# B&R Automation Studio project PickupStation
Automation Studio 4.12.4.107 SP; technology packages: mapp 5.23.1, mappCockpit 5.23.0, mappMotion 5.23.1, mappView 5.23.0

## Configuration Configuration

CPU X20CP1686X, AutomationRuntime H4.93, Build 4.1.2, Vc V4.73.0

### Task classes (Cpu.sw)
```
Cyclic#1:
  RSModelPic <- RSModelPick.prg
  ConveyorPr <- Source.Conveyor.ConveyorProgram.prg
  StamperPro <- Source.Stamper.StamperProgram.prg
Cyclic#2 (cycle 12000 us, tolerance 12000 us):
  MasterProg <- Source.Master.MasterProgram.prg
  MainMachin <- Source.MainMachine.MainMachineProgram.prg
  PusherProg <- Source.Pusher.PusherProgram.prg
  PickerProg <- Source.Picker.PickerProgram.prg
Cyclic#4:
  Alarms <- Source.Infrastructure.Alarms.Alarms.prg
  HMIProgram <- Source.HMI.HMIProgram.prg
DataObjects: McAcpSys
NcDataObjects: McDriveLog
Binaries: TCLang, McAcpDrv, udbdef, McAcpSim, mvLoader, arflatprv, mCoWebSc, TCData, FWRules, arcoal, arsvcreg, OpcUaSrv, Settings, iomap, asfw, Role, ashwac, sysconf, AxisConfig, arconfig, AlarmsCore, AlarmsHist, TC, ashwd, User, Cam, Users
Libraries: McBase, MpAxis, McAxis, MpBase, McAcpAx, CoTrace, AsZip, FileIO, runtime, MpAlarmX, astime, standard, asstring, MpServer, MpFile, MpUserX, asieccon, asbrstr, dataobj, asepl, asusb, aruser, arssl, sys_lib, powerlnk, arcert, ashw, aseth
```

### Hardware
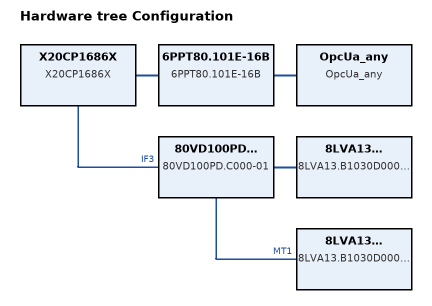
```
6PPT80.101E-16B : 6PPT80.101E-16B v1.0.6.0  [ETH1 -> X20CP1686X.IF2 [Cable Type=PowerlinkCable, Length=10, Version=1.0.0.3]; ETH2 -> OpcUa_any.ETH1 [Cable Type=PowerlinkCable, Length=10, Version=1.0.0.3]]
  Terminal = true
  Startmode = 2
  Mode = Manual
  InternetAddress = 192.168.0.2
  Subnetmask = 255.255.255.0
  ScreenRotation = 180
  PasswordVNC = 
  SelectedFavoriteWeb = 192.168.0.1:81
  BrowserVKeyboard = 0
  PasswordCIFS = 
  PasswordService = 
80VD100PD.C000-01 : 80VD100PD.C000-01 v2.5.0.0  [PLK1 -> X20CP1686X.IF3 (NodeNumber=1) [Cable Type=PowerlinkCable, Length=10, Version=1.0.0.3]; MT2 -> 8LVA13.B1030D000-0.MT]
  DriveConfiguration/Module:
    McAcoposTypeID = AcoposMicroDConfig
    ActivateACOPOSSimulationOnPLC = 1
  DriveConfiguration/Channel[1]/RealAxis:
    AxisReference = gAxisConveyorMpLink
    MechanicalElementsIsInvisible = 0
  DriveConfiguration/Channel[1]/RealAxis/MechanicalElements/Gearbox:
    InputIsReadOnly = 0
    Input = 1
    OutputIsReadOnly = 0
    Output = 1
  DriveConfiguration/Channel[1]/RealAxis/MechanicalElements/RotaryToLinearTransformation:
    ReferenceDistanceIsReadOnly = 0
    ReferenceDistance = 1
  DriveConfiguration/Channel[1]/RealAxis/Controller:
    ModeIsReadOnly = 0
    Mode = PositionController
  DriveConfiguration/Channel[1]/RealAxis/Controller/Mode/Position:
    ProportionalGain = 50.0
    IntegrationTime = 0.0
    PredictionTime = 0.0004
    TotalDelayTime = 0.0004
  DriveConfiguration/Channel[1]/RealAxis/Controller/Mode/Speed:
    ProportionalGainIsReadOnly = 0
    ProportionalGain = 2.0
    IntegrationTimeIsReadOnly = 0
    IntegrationTime = 0.0
    FilterTimeIsReadOnly = 0
    FilterTime = 0.0
  DriveConfiguration/Channel[1]/RealAxis/Controller/Mode/LoopFilters:
    LoopFilterXIsReadOnly = 0
    LoopFilter1 = NotUsed
    LoopFilter2 = NotUsed
    LoopFilter3 = NotUsed
  DriveConfiguration/Channel[1]/RealAxis/Homing:
    ModeIsReadOnly = 0
    Mode = Direct
  DriveConfiguration/Channel[1]/RealAxis/Homing/Mode:
    Position = 0.0
    ReferencePulse = NotUsed
  DriveConfiguration/Channel[1]/RealAxis/Homing:
    RestorePositionVariable = 
  DriveConfiguration/Channel[1]/RealAxis/StopReaction:
    QuickstopIsReadOnly = 0
    Quickstop = DecelerationLimit
    DriveErrorIsReadOnly = 0
    DriveError = DecelerationLimit
  DriveConfiguration/Channel[1]/RealAxis/MovementErrorLimits:
    PositionError = 1.0
    VelocityErrorMonitoring = Automatic1
  DriveConfiguration/Channel[1]/RealAxis:
    JerkFilterIsReadOnly = 0
    JerkFilter = NotUsed
    ZeroVibrationFilter = NotUsed
  DriveConfiguration/Channel[1]/RealAxis/DigitalInputs/HomingSwitch:
    SourceIsReadOnly = 0
    Source = NotUsed
    Level = High
  DriveConfiguration/Channel[1]/RealAxis/DigitalInputs/PositiveLimitSwitch:
    SourceIsReadOnly = 0
    Source = NotUsed
    Level = High
  DriveConfiguration/Channel[1]/RealAxis/DigitalInputs/NegativeLimitSwitch:
    SourceIsReadOnly = 0
    Source = NotUsed
    Level = High
  DriveConfiguration/Channel[1]/RealAxis/DigitalInputs/Trigger1:
    Source = X2Trigger1
    Level = High
  DriveConfiguration/Channel[1]/RealAxis/DigitalInputs/Trigger2:
    Source = X2Trigger2
    Level = High
  DriveConfiguration/Channel[1]/RealAxis/DigitalInputs/Quickstop:
    Input = NotUsed
  DriveConfiguration/Channel[1]/RealAxis/Simulation:
    SimulationModeOnPLC = SetValueGeneration
    SimulationModeOnACOPOS = NotUsed
  DriveConfiguration/Channel[2]/RealAxis:
    AxisReference = gAxisStamperMpLink
    MechanicalElementsIsInvisible = 0
  DriveConfiguration/Channel[2]/RealAxis/MechanicalElements/Gearbox:
    InputIsReadOnly = 0
    Input = 1
    OutputIsReadOnly = 0
    Output = 1
  DriveConfiguration/Channel[2]/RealAxis/MechanicalElements/RotaryToLinearTransformation:
    ReferenceDistanceIsReadOnly = 0
    ReferenceDistance = 1
  DriveConfiguration/Channel[2]/RealAxis/Controller:
    ModeIsReadOnly = 0
    Mode = PositionController
  DriveConfiguration/Channel[2]/RealAxis/Controller/Mode/Position:
    ProportionalGain = 50.0
    IntegrationTime = 0.0
    PredictionTime = 0.0004
    TotalDelayTime = 0.0004
  DriveConfiguration/Channel[2]/RealAxis/Controller/Mode/Speed:
    ProportionalGainIsReadOnly = 0
    ProportionalGain = 2.0
    IntegrationTimeIsReadOnly = 0
    IntegrationTime = 0.0
    FilterTimeIsReadOnly = 0
    FilterTime = 0.0
  DriveConfiguration/Channel[2]/RealAxis/Controller/Mode/LoopFilters:
    LoopFilterXIsReadOnly = 0
    LoopFilter1 = NotUsed
    LoopFilter2 = NotUsed
    LoopFilter3 = NotUsed
  DriveConfiguration/Channel[2]/RealAxis/Homing:
    ModeIsReadOnly = 0
    Mode = Direct
  DriveConfiguration/Channel[2]/RealAxis/Homing/Mode:
    Position = 0.0
    ReferencePulse = NotUsed
  DriveConfiguration/Channel[2]/RealAxis/Homing:
    RestorePositionVariable = 
  DriveConfiguration/Channel[2]/RealAxis/StopReaction:
    QuickstopIsReadOnly = 0
    Quickstop = DecelerationLimit
    DriveErrorIsReadOnly = 0
    DriveError = DecelerationLimit
  DriveConfiguration/Channel[2]/RealAxis/MovementErrorLimits:
    PositionError = 1.0
    VelocityErrorMonitoring = Automatic1
  DriveConfiguration/Channel[2]/RealAxis:
    JerkFilterIsReadOnly = 0
    JerkFilter = NotUsed
    ZeroVibrationFilter = NotUsed
  DriveConfiguration/Channel[2]/RealAxis/DigitalInputs/HomingSwitch:
    SourceIsReadOnly = 0
    Source = NotUsed
    Level = High
  DriveConfiguration/Channel[2]/RealAxis/DigitalInputs/PositiveLimitSwitch:
    SourceIsReadOnly = 0
    Source = NotUsed
    Level = High
  DriveConfiguration/Channel[2]/RealAxis/DigitalInputs/NegativeLimitSwitch:
    SourceIsReadOnly = 0
    Source = NotUsed
    Level = High
  DriveConfiguration/Channel[2]/RealAxis/DigitalInputs/Trigger1:
    Source = X2Trigger1
    Level = High
  DriveConfiguration/Channel[2]/RealAxis/DigitalInputs/Trigger2:
    Source = X2Trigger2
    Level = High
  DriveConfiguration/Channel[2]/RealAxis/DigitalInputs/Quickstop:
    Input = NotUsed
  DriveConfiguration/Channel[2]/RealAxis/Simulation:
    SimulationModeOnPLC = SetValueGeneration
    SimulationModeOnACOPOS = NotUsed
  DriveConfiguration/Channel[2]/RealAxis/AxisFeatures:
    FeatureRef[1] = CamAutomat
8LVA13.B1030D000-0 : 8LVA13.B1030D000-0 v2.2.0.3  [MT -> 80VD100PD.C000-01.MT2]
  M1/MotorParameters:
    MOTOR_AMB_TEMP_RATED = 40
8LVA13.B1030D000-0a : 8LVA13.B1030D000-0 v2.2.0.3  [MT -> 80VD100PD.C000-01.MT1]
  M1/MotorParameters:
    MOTOR_AMB_TEMP_RATED = 40
OpcUa_any : OpcUa_any v1.0.0.1  [ETH1 -> 6PPT80.101E-16B.ETH2 [Cable Type=PowerlinkCable, Length=10, Version=1.0.0.3]]
  ServerEndpointUrl = opc.tcp://192.168.0.3:4840
  Channel1
  ChannelID1 = OUT_HeartBeat
  ChannelBrowsePath1 = /0:Root/0:Objects/4:PLC/4:Modules/6:&:&:/6:Global PV/6:gPickingStation/6:Outputs/6:HeartBeat
  ChannelDirection1 = OUT
  ChannelSamplingInterval1 = 50
  Channel2
  ChannelID2 = OUT_Error
  ChannelBrowsePath2 = /0:Root/0:Objects/4:PLC/4:Modules/6:&:&:/6:Global PV/6:gPickingStation/6:Outputs/6:Error
  ChannelDirection2 = OUT
  ChannelSamplingInterval2 = 50
  Channel3
  ChannelID3 = OUT_WaitingStart
  ChannelBrowsePath3 = /0:Root/0:Objects/4:PLC/4:Modules/6:&:&:/6:Global PV/6:gPickingStation/6:Outputs/6:WaitingStart
  ChannelDirection3 = OUT
  ChannelSamplingInterval3 = 50
  Channel4
  ChannelID4 = OUT_WaitingModeSelection
  ChannelBrowsePath4 = /0:Root/0:Objects/4:PLC/4:Modules/6:&:&:/6:Global PV/6:gPickingStation/6:Outputs/6:WaitingModeSelection
  ChannelDirection4 = OUT
  ChannelSamplingInterval4 = 50
  Channel5
  ChannelID5 = OUT_WaitingInit
  ChannelBrowsePath5 = /0:Root/0:Objects/4:PLC/4:Modules/6:&:&:/6:Global PV/6:gPickingStation/6:Outputs/6:WaitingInit
  ChannelDirection5 = OUT
  ChannelSamplingInterval5 = 50
  Channel6
  ChannelID6 = OUT_InitDone
  ChannelBrowsePath6 = /0:Root/0:Objects/4:PLC/4:Modules/6:&:&:/6:Global PV/6:gPickingStation/6:Outputs/6:InitDone
  ChannelDirection6 = OUT
  ChannelSamplingInterval6 = 50
  Channel7
  ChannelID7 = OUT_Started
  ChannelBrowsePath7 = /0:Root/0:Objects/4:PLC/4:Modules/6:&:&:/6:Global PV/6:gPickingStation/6:Outputs/6:Started
  ChannelDirection7 = OUT
  ChannelSamplingInterval7 = 50
  Channel8
  ChannelID8 = OUT_ClearStatsDone
  ChannelBrowsePath8 = /0:Root/0:Objects/4:PLC/4:Modules/6:&:&:/6:Global PV/6:gPickingStation/6:Outputs/6:ClearStatsDone
  ChannelDirection8 = OUT
  ChannelSamplingInterval8 = 50
  Channel9
  ChannelID9 = OUT_LinkActive
  ChannelBrowsePath9 = /0:Root/0:Objects/4:PLC/4:Modules/6:&:&:/6:Global PV/6:gPickingStation/6:Outputs/6:LinkActive
  ChannelDirection9 = OUT
  ChannelSamplingInterval9 = 50
  Channel10
  ChannelID10 = OUT_ActStampOffset
  ChannelBrowsePath10 = /0:Root/0:Objects/4:PLC/4:Modules/6:&:&:/6:Global PV/6:gPickingStation/6:Outputs/6:ActStampOffset
  ChannelDirection10 = OUT
  ChannelSamplingInterval10 = 50
  ChannelType10 = REAL
  Channel11
  ChannelID11 = OUT_ActStampIncluded
  ChannelBrowsePath11 = /0:Root/0:Objects/4:PLC/4:Modules/6:&:&:/6:Global PV/6:gPickingStation/6:Outputs/6:ActStampIncluded
  ChannelDirection11 = OUT
  ChannelSamplingInterval11 = 50
  Channel12
  ChannelID12 = OUT_CapsOnConveyor
  ChannelBrowsePath12 = /0:Root/0:Objects/4:PLC/4:Modules/6:&:&:/6:Global PV/6:gPickingStation/6:Outputs/6:CapsOnConveyor
  ChannelDirection12 = OUT
  ChannelSamplingInterval12 = 50
  ChannelType12 = USINT
  Channel13
  ChannelID13 = IN_HeartBeat
  ChannelBrowsePath13 = /0:Root/0:Objects/4:PLC/4:Modules/6:&:&:/6:Global PV/6:gPickingStation/6:Inputs/6:HeartBeat
  ChannelPublishingInterval13 = 50
  Channel14
  ChannelID14 = IN_Reset
  ChannelBrowsePath14 = /0:Root/0:Objects/4:PLC/4:Modules/6:&:&:/6:Global PV/6:gPickingStation/6:Inputs/6:Reset
  ChannelPublishingInterval14 = 50
  Channel15
  ChannelID15 = IN_Error
  ChannelBrowsePath15 = /0:Root/0:Objects/4:PLC/4:Modules/6:&:&:/6:Global PV/6:gPickingStation/6:Inputs/6:Error
  ChannelPublishingInterval15 = 50
  Channel16
  ChannelID16 = IN_ClearStats
  ChannelBrowsePath16 = /0:Root/0:Objects/4:PLC/4:Modules/6:&:&:/6:Global PV/6:gPickingStation/6:Inputs/6:ClearStats
  ChannelPublishingInterval16 = 50
  Channel17
  ChannelID17 = IN_Init
  ChannelBrowsePath17 = /0:Root/0:Objects/4:PLC/4:Modules/6:&:&:/6:Global PV/6:gPickingStation/6:Inputs/6:Init
  ChannelPublishingInterval17 = 50
  Channel18
  ChannelID18 = IN_Start
  ChannelBrowsePath18 = /0:Root/0:Objects/4:PLC/4:Modules/6:&:&:/6:Global PV/6:gPickingStation/6:Inputs/6:Start
  ChannelPublishingInterval18 = 50
  Channel19
  ChannelID19 = IN_AutomaticMode
  ChannelBrowsePath19 = /0:Root/0:Objects/4:PLC/4:Modules/6:&:&:/6:Global PV/6:gPickingStation/6:Inputs/6:AutomaticMode
  ChannelPublishingInterval19 = 50
  Channel20
  ChannelID20 = IN_StampIncluded
  ChannelBrowsePath20 = /0:Root/0:Objects/4:PLC/4:Modules/6:&:&:/6:Global PV/6:gPickingStation/6:Inputs/6:StampIncluded
  ChannelPublishingInterval20 = 50
  Channel21
  ChannelID21 = IN_StampOffset
  ChannelBrowsePath21 = /0:Root/0:Objects/4:PLC/4:Modules/6:&:&:/6:Global PV/6:gPickingStation/6:Inputs/6:StampOffset
  ChannelPublishingInterval21 = 50
  ChannelType21 = REAL
  Channel22
  ChannelID22 = IN_ConveyorSpeed
  ChannelBrowsePath22 = /0:Root/0:Objects/4:PLC/4:Modules/6:&:&:/6:Global PV/6:gPickingStation/6:Inputs/6:ConveyorSpeed
  ChannelPublishingInterval22 = 50
  ChannelType22 = REAL
X20CP1686X : X20CP1686X v1.8.0.0
  Connector IF2:
    ActivateDevice = 1
    Mode = Manual
    InternetAddress = 192.168.0.1
    SubnetMask = 255.255.255.0
    ActivateSnmp = 2
  ConfigurationID = PickupStation_Configuration
  VolatileGlobalPvSize = 125535
  TimerDeviceType = EPLX2X
  TimerDevice = X20CP1686X.IF3
  Cyclic1Tolerance = 0
  Cyclic2Duration = 12000
  Cyclic2Tolerance = 12000
  FileDevice1
  FileDeviceName1 = USER
  FileDevicePath1 = USER_PATH
  ActivateOpcUa = 1
  OpcUaInformationModels_PV_Version = 2
  OpcUaInformationModel_Facet = 0
  OpcUaInformationModel_TypeInformation = 0
  OpcUaInformationModel_BaseObjectTypeForStructures = 0
```

### IoMap.iom - X20CP1686X/IoMap.iom
```iecst
VAR_CONFIG
	Cyclic#2.::gMaster.Outputs.HeartBeat AT %IX."OpcUa_any".IN_HeartBeat;
	Cyclic#2.::gMaster.Inputs.HeartBeat AT %QX."OpcUa_any".OUT_HeartBeat;
	Cyclic#2.::gMaster.Inputs.Error AT %QX."OpcUa_any".OUT_Error;
	Cyclic#2.::gMaster.Inputs.WaitingStart AT %QX."OpcUa_any".OUT_WaitingStart;
	Cyclic#2.::gMaster.Inputs.WaitingModeSelection AT %QX."OpcUa_any".OUT_WaitingModeSelection;
	Cyclic#2.::gMaster.Inputs.WaitingInit AT %QX."OpcUa_any".OUT_WaitingInit;
	Cyclic#2.::gMaster.Inputs.InitDone AT %QX."OpcUa_any".OUT_InitDone;
	Cyclic#2.::gMaster.Inputs.Started AT %QX."OpcUa_any".OUT_Started;
	Cyclic#2.::gMaster.Inputs.ClearStatsDone AT %QX."OpcUa_any".OUT_ClearStatsDone;
	Cyclic#2.::gMaster.Outputs.Reset AT %IX."OpcUa_any".IN_Reset;
	Cyclic#2.::gMaster.Outputs.Error AT %IX."OpcUa_any".IN_Error;
	Cyclic#2.::gMaster.Outputs.ClearStats AT %IX."OpcUa_any".IN_ClearStats;
	Cyclic#2.::gMaster.Outputs.Init AT %IX."OpcUa_any".IN_Init;
	Cyclic#2.::gMaster.Outputs.Start AT %IX."OpcUa_any".IN_Start;
	Cyclic#2.::gMaster.Outputs.AutomaticMode AT %IX."OpcUa_any".IN_AutomaticMode;
	Cyclic#2.::gMaster.Outputs.StampIncluded AT %IX."OpcUa_any".IN_StampIncluded;
	Cyclic#2.::gMaster.Outputs.StampOffset AT %ID."OpcUa_any".IN_StampOffset;
	Cyclic#2.::gMaster.Outputs.ConveyorSpeed AT %ID."OpcUa_any".IN_ConveyorSpeed;
	Cyclic#2.::gMainMachine.Commands.OpcuaClientOk AT %IX."OpcUa_any".ModuleOk;
	Cyclic#2.::gMaster.Inputs.LinkActive AT %QX."OpcUa_any".OUT_LinkActive;
	Cyclic#2.::gMaster.Inputs.ActStampOffset AT %QD."OpcUa_any".OUT_ActStampOffset;
	Cyclic#2.::gMaster.Inputs.ActStampIncluded AT %QX."OpcUa_any".OUT_ActStampIncluded;
	::gMaster.Inputs.AskRemoveCaps AT %QX."OpcUa_any".OUT_AskRemoveCaps;
	Cyclic#2.::gMaster.Inputs.CapsOnConveyor AT %QB."OpcUa_any".OUT_CapsOnConveyor;
END_VAR
```

### AxisConfig.axis - X20CP1686X/mappMotion/AxisConfig.axis
```
Element gAxisConveyorMpLink (Type=axis)
  BaseTypeIsReadOnly = 0
  BaseType = LinearPeriodic
    MeasurementUnit = 5066068
    MeasurementResolutionIsReadOnly = 0
    MeasurementResolution = 0.01
    CountDirectionIsReadOnly = 0
    CountDirection = Standard
    PeriodSettings:
      Period = 580
  MovementLimitsIsReadOnly = 0
  MovementLimits = Internal
    Position:
      LowerLimitMin = -1.79769313486231E308
      UpperLimitMax = 1.79769313486231E308
      LowerLimit = -1000.0
      UpperLimit = 1000.0
    VelocityIsReadOnly = 0
    Velocity:
      VelocityMax = 3.4E38
      Velocity = 500
    AccelerationIsReadOnly = 0
    Acceleration:
      AccelerationMax = 3.4E38
      Acceleration = 5000
    DecelerationIsReadOnly = 0
    Deceleration:
      DecelerationMax = 3.4E38
      Deceleration = 5000
  Alarms = MpAlarmX
    mapp.AlarmX.Core.Configuration:
      [2]:
        Severity = 0
Element gAxisStamperMpLink (Type=axis)
  BaseTypeIsReadOnly = 0
  BaseType = Linear
    MeasurementUnit = 5066068
    MeasurementResolutionIsReadOnly = 0
    MeasurementResolution = 0.01
    CountDirectionIsReadOnly = 0
    CountDirection = Standard
  MovementLimitsIsReadOnly = 0
  MovementLimits = Internal
    Position:
      LowerLimitMin = -1.79769313486231E308
      UpperLimitMax = 1.79769313486231E308
      LowerLimit = 0
      UpperLimit = 0.46
    VelocityIsReadOnly = 0
    Velocity:
      VelocityMax = 3.4E38
      Velocity = 100000
    AccelerationIsReadOnly = 0
    Acceleration:
      AccelerationMax = 3.4E38
      Acceleration = 200000
    DecelerationIsReadOnly = 0
    Deceleration:
      DecelerationMax = 3.4E38
      Deceleration = 200000
  Alarms = MpAlarmX
    mapp.AlarmX.Core.Configuration:
      [2]:
        Severity = 0
```

### Cam.axisfeature - X20CP1686X/mappMotion/Cam.axisfeature
```
Element CamAutomat (Type=axisfeature)
  Type = CamAutomat
    CamAutomatType = ACOPOS
      CommonParameters:
        Master:
          ValueSource = SetPosition
            AxisReference = gAxisConveyorMpLink
            MaxVelocity = 500
          StartPosition = 0.0
          StartInterval = MasterAxisPeriod
        AdvancedParameters:
          StartStateParameters:
            StartState = 0
            RelMasterStartPos = 0.0
          AdditiveAxes:
            AdditiveMasterValueSource = NotUsed
            AdditiveSlaveValueSource = NotUsed
          MasterStartPositionMode = NotEvaluatedAnew
          ControlSettings:
            CrossLeftBoundary = PositionLimitedHorizontal
            CamChangeImmediately = CurrentMasterMoveDir
          MessageSettings:
            ErrorsInStandby = NoErrorMessages
          TriggerAndLatch:
            Trigger1Delay = 0.0
            Trigger2Delay = 0.0
            SlaveLatchParID = 0
          EventParIDs
          StartIntervals
          Factors:
            SlaveFactorParID = 0
      States:
        State0 = Used
          Events:
            Event[0]:
              Type = Signal1FromPLC
              Transition = Immediately
              SynchronousUpdate = NotUsed
              NextState = 1
        State[1]:
          Cam = Predefined
            PredefinedCam = OneToOne
          MasterFactor = 20000
          SlaveFactor = 20000
          CompensationMode = DistancesBetweenExitEntryPoints
            MasterDistance = 100
            SlaveDistance = 20
            AdvancedParameters = NotUsed
          AdvancedParameters:
            RepeatCounterInit = 0
            MasterValueSource = CommonMaster
          Events:
            Event[0]:
              Type = StateEnd
              Transition = Immediately
              SynchronousUpdate = NotUsed
              NextState = 2
        State[2]:
          Cam = Predefined
            PredefinedCam = ZeroPoint
          MasterFactor = 1
          SlaveFactor = 0
          CompensationMode = DistancesBetweenExitEntryPoints
            MasterDistance = 100
            SlaveDistance = -220
            AdvancedParameters = NotUsed
          AdvancedParameters:
            RepeatCounterInit = 0
            MasterValueSource = CommonMaster
          Events:
            Event[0]:
              Type = StateEnd
              Transition = Immediately
              SynchronousUpdate = NotUsed
              NextState = 0
```

- Safety project (password-protected, skipped)

### AlarmsCore.mpalarmxcore - X20CP1686X/mappServices/AlarmsCore.mpalarmxcore
```
Element gAlarmXCoreMpLink (Type=mpalarmxcore)
  mapp.AlarmX.Core:
    Mapping:
      [0]
    BySeverity:
      [0]:
        Severity = 1
        [0] = Reaction
          Name = STOP
  mapp.AlarmX.Core.Configuration:
    [0]:
      Name = PickerTimeoutForward
      Message = {$Source/Picker/Alarms/PickerTimeoutForward}
    [1]:
      Name = PickerTimeoutBackward
      Message = {$Source/Picker/Alarms/PickerTimeoutBackward}
    [2]:
      Name = PickerTimeoutVacuumPick
      Message = {$Source/Picker/Alarms/PickerTimeoutVacuumPick}
    [3]:
      Name = PickerTimeoutVacuumPlace
      Message = {$Source/Picker/Alarms/PickerTimeoutVacuumPlace}
    [4]:
      Name = PickerInvalidSensorsCombination
      Message = {$Source/Picker/Alarms/PickerInvalidSensorsCombination}
      Behavior = PersistentAlarm
    [5]:
      Name = PusherTimeoutForward
      Message = {$Source/Pusher/Alarms/PusherTimeoutForward}
    [6]:
      Name = PusherTimeoutBackward
      Message = {$Source/Pusher/Alarms/PusherTimeoutBackward}
    [7]:
      Name = PusherTimeoutMagazineEmpty
      Message = {$Source/Pusher/Alarms/PusherTimeoutMagazineEmpty}
    [8]:
      Name = PusherInvalidSensorsCombination
      Message = {$Source/Pusher/Alarms/PusherInvalidSensorsCombination}
      Behavior = PersistentAlarm
    [9]:
      Name = ConveyorTimeoutHoming
      Message = {$Source/Conveyor/Alarms/ConveyorTimeoutHoming}
    [10]:
      Name = ConveyorTimeoutPowerOn
      Message = {$Source/Conveyor/Alarms/ConveyorTimeoutPowerOn}
    [11]:
      Name = ConveyorMissedCap
      Message = {$Source/Conveyor/Alarms/ConveyorMissedCap}
    [12]:
      Name = ConveyorAxisError
      Message = {$Source/Conveyor/Alarms/ConveyorAxisError}
      Behavior = PersistentAlarm
    [13]:
      Name = ConveyorInitFail
      Message = {$Source/Conveyor/Alarms/ConveyorInitFail}
    [14]:
      Name = ConveyorTooManyCaps
      Message = {$Source/Conveyor/Alarms/ConveyorTooManyCaps}
      Behavior = PersistentAlarm
    [15]:
      Name = StamperAxisError
      Message = {$Source/Stamper/Alarms/StamperAxisError}
      Behavior = PersistentAlarm
    [16]:
      Name = StamperInvalidSensorsCombination
      Message = {$Source/Stamper/Alarms/StamperInvalidSensorsCombination}
      Behavior = PersistentAlarm
    [17]:
      Name = StamperTimeoutHoming
      Message = {$Source/Stamper/Alarms/StamperTimeoutHoming}
    [18]:
      Name = StamperTimeoutPowerOn
      Message = {$Source/Stamper/Alarms/StamperTimeoutPowerOn}
    [19]:
      Name = StamperTimeoutStampBackward
      Message = {$Source/Stamper/Alarms/StamperTimeoutStampBackward}
    [20]:
      Name = StamperTimeoutStampForward
      Message = {$Source/Stamper/Alarms/StamperTimeoutStampForward}
    [21]:
      Name = StamperAxisTimeout
      Message = {$Source/Stamper/Alarms/StamperAxisTimeout}
    [22]:
      Name = MainMachineEmergencyCircuitInterrupted
      Message = {$Source/MainMachine/Alarms/MainMachineEmergencyCircuitInterrupted}
      Behavior = PersistentAlarm
    [23]:
      Name = MainMachineCommunicationLost
      Message = {$Source/MainMachine/Alarms/MainMachineCommunicationLost}
      Behavior = PersistentAlarm
    [24]:
      Name = MainMachineInitializationTimeout
      Message = {$Source/MainMachine/Alarms/MainMachineInitializationTimeout}
    [25]:
      Name = MasterInError
      Message = {$Source/Master/Alarms/MasterInError}
      Behavior:
        MultipleInstances = FALSE
```

### AlarmsHist.mpalarmxhistory - X20CP1686X/mappServices/AlarmsHist.mpalarmxhistory
```
Element gAlarmXHistoryMpLink (Type=mpalarmxhistory)
```

### Users.mpuserx - X20CP1686X/mappServices/Users.mpuserx
```
Element UserMgmtX (Type=mpuserx)
  Mgr:
    LoginAttempts = 0
  ServerSettings:
    Server:
      AdditionalUserData:
        [0] = mail
        [1] = telephoneNumber
  Users:
    DefUser#1:
      id = admin
      name = Andrea Pennisi
      lang = it
      unit = imperial
    DefUser#2:
      id = Anonymous
      lang = en
      unit = metric
  Groups:
    DefGroup#1:
      id = Everyone
      level = 0
    DefGroup#2:
      id = Administrators
      admin = TRUE
```

## Logical view

Binary libraries used (declarations not repeated): operator, runtime, astime, AsIecCon, McBase 5.23.1, MpAxis 5.23.1, McAxis 5.23.1, MpBase 5.23.0, McAcpAx 5.23.1, CoTrace 5.23.0, AsZip, FileIO, MpAlarmX 5.23.1, standard, asstring, MpServer 5.23.0, MpFile 5.23.1, MpUserX 5.23.1


### Program Logical/RSModelPick (IEC) - IO Interface to the RobotStudio model (Pickup IOs)

#### Main.st - Init, cyclic, exit code
```iecst
PROGRAM _INIT
	aiLogoAxisActPos;
	diMagazineEmpty;
	diCapAtPickup;
	diCapPusherForward;
	diCapPusherBack;
	diPickupArmBack;
	diPickupArmForward;
	diCapGripperVacuum;
	diCapOnLogoConveyor;
	diCapExitLogoConveyor;
	diLogoStamperBack;
	diLogoStamperForward;
	aoLogoConveyorSetSpeed;
	doCapPusher;
	doPickupArmForward;
	doPickupArmBack;
	doCapGripperPick;
	aoLogoAxisSetPos;
	doLogoStamper;
	doLogoConveyorClear;

END_PROGRAM

PROGRAM _CYCLIC
	// Pusher
	gPusher.Interface.Inputs.PusherInForwardPosition := diCapPusherForward;
	gPusher.Interface.Inputs.PusherInBackwardPosition := diCapPusherBack;
	gPusher.Interface.Inputs.CapAtPickPosition := diCapAtPickup;
	gPusher.Interface.Inputs.MagazineEmpty := diMagazineEmpty;

	doCapPusher := gPusher.Interface.Outputs.MoveForward;

	// Picker
	gPicker.Interface.Inputs.ArmForward := diPickupArmForward;
	gPicker.Interface.Inputs.ArmBackward := diPickupArmBack;
	gPicker.Interface.Inputs.GripperVacuum := diCapGripperVacuum;

	doPickupArmForward := gPicker.Interface.Outputs.ArmForward;
	doPickupArmBack := gPicker.Interface.Outputs.ArmBackward;
	doCapGripperPick := gPicker.Interface.Outputs.GripperPick;

	// Conveyor
	gConveyor.Interface.Inputs.CapInStartPosition := diCapOnLogoConveyor;
	gConveyor.Interface.Inputs.CapInExitPosition := diCapExitLogoConveyor;

	aoLogoConveyorSetSpeed := gConveyor.Interface.Outputs.SetSpeed/1000;

	// Stamper
	gStamper.Interface.Inputs.ActualPosition := aiLogoAxisActPos*1000;
	gStamper.Interface.Inputs.StampIsForward := diLogoStamperForward;
	gStamper.Interface.Inputs.StampIsBackward := diLogoStamperBack;

	aoLogoAxisSetPos := LREAL_TO_REAL(gStamper.Interface.Outputs.SetPosition/1000);
	doLogoStamper := gStamper.Interface.Outputs.StampForward;
END_PROGRAM

PROGRAM _EXIT

END_PROGRAM
```

#### Variables.var - Local variables
```iecst
(*Inputs*)
VAR
	diMagazineEmpty : BOOL := 0;
	diCapAtPickup : BOOL := 0;
	diCapPusherForward : BOOL := 0;
	diCapPusherBack : BOOL := 0;
	diPickupArmForward : BOOL := 0;
	diPickupArmBack : BOOL := 0;
	diCapGripperVacuum : BOOL := 0;
	diCapOnLogoConveyor : BOOL := 0;
	diLogoStamperForward : BOOL := 0;
	diLogoStamperBack : BOOL := 0;
	diCapExitLogoConveyor : BOOL := 0;
	aiLogoAxisActPos : REAL := 0.0; (*[m]*)
END_VAR
(*Outputs*)
VAR
	doCapPusher : BOOL := 0;
	doPickupArmForward : BOOL := 0;
	doPickupArmBack : BOOL := 0;
	doCapGripperPick : BOOL := 0;
	doLogoStamper : BOOL := 0;
	aoLogoConveyorSetSpeed : REAL := 0.0; (*[m/s]*)
	aoLogoAxisSetPos : REAL := 0.0; (*[m]*)
END_VAR
(*Model Interaction*)
VAR
	doLogoConveyorClear : BOOL := 0;
END_VAR
```

### AlarmsGlobalVariables.var
```iecst
VAR
	gAlarms : AlarmsType;
END_VAR
```

### AlarmsGlobalTypes.typ
```iecst
TYPE
	AlarmsType : 	STRUCT
		Feedbacks : AlarmsFeedbacksType;
		MpAlarmXListUIConnect : MpAlarmXListUIConnectType;
	END_STRUCT;
	AlarmsFeedbacksType : 	STRUCT
		Pendings : UDINT;
	END_STRUCT;
END_TYPE
```

### Program Logical/Source/Infrastructure/Alarms/Alarms (IEC)

#### Main.st - Init, cyclic, exit code
```iecst
PROGRAM _INIT
	// This program is used to manage the machine alarms. Alarms are set/reset in the modules.

	MpAlarmXCoreFB(MpLink := ADR(gAlarmXCoreMpLink), Enable := TRUE);

	MpAlarmXHistoryFB(MpLink := ADR(gAlarmXHistoryMpLink), Enable := TRUE, DeviceName := ADR('ALARMS'));

	MpAlarmXListUIFB(MpLink :=  ADR(gAlarmXCoreMpLink), Enable := TRUE, UIConnect := ADR(gAlarms.MpAlarmXListUIConnect));

END_PROGRAM

PROGRAM _CYCLIC
	MpAlarmXCoreFB();

	MpAlarmXHistoryFB();

	MpAlarmXListUIFB();

	gAlarms.Feedbacks.Pendings := MpAlarmXCoreFB.PendingAlarms;
END_PROGRAM

PROGRAM _EXIT
	MpAlarmXCoreFB.Enable := FALSE;
	MpAlarmXCoreFB();

	MpAlarmXHistoryFB.Enable := FALSE;
	MpAlarmXHistoryFB();

	MpAlarmXListUIFB.Enable := FALSE;
	MpAlarmXListUIFB();

END_PROGRAM
```

#### Variables.var - Local variables
```iecst
VAR
	MpAlarmXCoreFB : MpAlarmXCore;
	MpAlarmXHistoryFB : MpAlarmXHistory;
	MpAlarmXListUIFB : MpAlarmXListUI;
END_VAR
```

### PusherGlobalTypes.typ
```iecst
TYPE
	PusherType : 	STRUCT  (*Pusher Main type*)
		Commands : PusherCommandsType;
		Feedbacks : PusherFeedbacksType;
		Interface : PusherInterfaceType;
	END_STRUCT;
	PusherCommandsType : 	STRUCT
		Enable : BOOL;
		Reset : BOOL;
		Automatic : PusherAutomaticCommandsType;
		Manual : PusherManualCommandsType;
	END_STRUCT;
	PusherFeedbacksType : 	STRUCT  (*Pusher Feedbacks type*)
		Enabled : BOOL;
		Error : BOOL;
		WaitingStart : BOOL;
		CapReady : BOOL;
		WaitingTakeACapCommand : BOOL;
		InitDone : BOOL;
		InitPosition : BOOL;
		TakeACapDone : BOOL;
	END_STRUCT;
	PusherInterfaceType : 	STRUCT  (*Pusher Interface type*)
		Inputs : PusherInterfaceInputsType;
		Outputs : PusherInterfaceOutputsType;
	END_STRUCT;
	PusherInterfaceOutputsType : 	STRUCT  (*Pusher Interface Output type*)
		MoveForward : BOOL;
	END_STRUCT;
	PusherInterfaceInputsType : 	STRUCT  (*Pusher Interface Input type*)
		PusherInBackwardPosition : BOOL;
		PusherInForwardPosition : BOOL;
		CapAtPickPosition : BOOL;
		MagazineEmpty : BOOL;
	END_STRUCT;
	PusherManualCommandsType : 	STRUCT
		Enable : BOOL;
		Push : BOOL;
	END_STRUCT;
	PusherAutomaticCommandsType : 	STRUCT
		Start : BOOL;
		Init : BOOL;
		TakeACap : BOOL;
	END_STRUCT;
END_TYPE
```

### PusherGlobalVariables.var
```iecst
VAR
    gPusher : PusherType;
END_VAR
```

### Program Logical/Source/Pusher/PusherProgram (IEC)

#### Main.st - Init, cyclic, exit code
```iecst
//******************************************************************************************************
// Program: 	PusherProgram
// Author: 		Andrea Pennisi
// Rev.: 		1.0.0
// Date:		5.12.2023
//
// Description:
// This module is used to pick a cap from the magazine station to the pick position.
// Only pneumatic motion in this module
//******************************************************************************************************

PROGRAM _INIT

    ResetOutputsAction;
    ResetFeedbacksAction;

    MachineState.NextState := WAITING_INIT;

END_PROGRAM

PROGRAM _CYCLIC

    // Enable module
    IF NOT gPusher.Commands.Enable THEN
        ResetOutputsAction;
		ResetFeedbacksAction;
		ResetAlarmsAction;
        RETURN;
	END_IF

	IF EDGENEG(gPusher.Commands.Automatic.Start) THEN
		IF MachineState.NextState <> ERROR THEN
			MachineState.NextState := WAITING_START;
		END_IF
	END_IF

	IF EDGEPOS(gPusher.Commands.Automatic.Init) THEN
		IF MachineState.NextState <> ERROR THEN
			MachineState.NextState := WAITING_INIT;
		END_IF
	END_IF

	// Alarms
	SetAlarmsAction;

    // Machine state
    MachineStateManagementAction;
    CASE MachineState.ActualState OF

		WAITING_INIT:
			MachineState.TimeoutTimer.PT := T#0S; // Timeout disabled in this state
			IF MachineState.NewTriggerState THEN
				ResetOutputsAction;
				gPusher.Feedbacks.TakeACapDone := FALSE;
			END_IF
			IF gPusher.Commands.Automatic.Init THEN
				MachineState.NextState := MOVE_BACKWARD;

			ELSIF gPusher.Commands.Manual.Enable THEN
				MachineState.NextState := MANUALS;

			END_IF

		MANUALS:
			MachineState.TimeoutTimer.PT := T#0S; // Timeout disabled in this state
			// Manual commands
			gPusher.Interface.Outputs.MoveForward := gPusher.Commands.Manual.Push;
			IF NOT gPusher.Commands.Manual.Enable THEN
				MachineState.NextState := WAITING_INIT;
			END_IF

		MOVE_BACKWARD:
			MachineState.TimeoutTimer.PT := T#3S;
			IF gPusher.Interface.Inputs.PusherInBackwardPosition THEN
				MachineState.NextState := WAITING_START;
			END_IF

		WAITING_START:
			MachineState.TimeoutTimer.PT := T#0S; // Timeout disabled in this state
			IF gPusher.Commands.Automatic.Start THEN
				MachineState.NextState := WAITING_MAGAZINE;

			ELSIF gPusher.Commands.Manual.Enable THEN
				MachineState.NextState := MANUALS;
			END_IF

		WAITING_MAGAZINE:
			MachineState.TimeoutTimer.PT := T#3S;
			IF NOT gPusher.Interface.Inputs.MagazineEmpty THEN
				MachineState.NextState := WAITING_TAKE_A_CAP_COMMAND;
			END_IF

		WAITING_TAKE_A_CAP_COMMAND:
			MachineState.TimeoutTimer.PT := T#0S; // Timeout disabled in this state
			IF NOT gPusher.Interface.Inputs.CapAtPickPosition AND gPusher.Commands.Automatic.TakeACap THEN
				gPusher.Feedbacks.TakeACapDone := FALSE;
				MachineState.NextState := MOVE_FORWARD;
			END_IF

		MOVE_FORWARD:
			MachineState.TimeoutTimer.PT := T#3S;
			gPusher.Interface.Outputs.MoveForward := TRUE;
			IF gPusher.Interface.Inputs.CapAtPickPosition THEN
				gPusher.Interface.Outputs.MoveForward := FALSE;
				gPusher.Feedbacks.TakeACapDone := TRUE;
				MachineState.NextState := MOVE_BACKWARD;
			END_IF

        ERROR:
			MachineState.TimeoutTimer.PT := T#0S; // Timeout disabled in this state
			ResetOutputsAction;
			IF NOT Internal.Error THEN
				MachineState.NextState := WAITING_INIT;
			END_IF

        ELSE
            MachineState.NextState := WAITING_INIT;

    END_CASE

    FeedbacksUpdateAction;

END_PROGRAM

PROGRAM _EXIT

END_PROGRAM
```

#### Types.typ - Local data types
```iecst
TYPE
	MachineStateType : 	STRUCT  (*Machine state main type*)
		OldState : MachineStateEnum; (*Actual state*)
		ActualState : MachineStateEnum; (*Actual state*)
		NextState : MachineStateEnum; (*Next state*)
		NewTriggerState : BOOL; (*Trigger state change*)
		TimeoutTimer : TON; (*State timeout*)
	END_STRUCT;
	MachineStateEnum :
		( (*Machine State enumeration*)
		WAITING_INIT, (*WAITING state*)
		MANUALS,
		WAITING_START, (*WAITING state*)
		MOVE_BACKWARD,
		WAITING_MAGAZINE, (*ERROR state*)
		WAITING_TAKE_A_CAP_COMMAND,
		MOVE_FORWARD,
		ERROR
		);
	InternalType : 	STRUCT
		Error : BOOL;
	END_STRUCT;
END_TYPE
```

#### Variables.var - Local variables
```iecst
VAR
	MachineState : MachineStateType;
	Internal : InternalType;
END_VAR
```

#### Actions.st
```iecst
ACTION FeedbacksUpdateAction:

	gPusher.Feedbacks.Enabled := TRUE;
    gPusher.Feedbacks.WaitingStart := MachineState.ActualState = WAITING_START;
	gPusher.Feedbacks.Error := MachineState.ActualState = ERROR;
	gPusher.Feedbacks.WaitingTakeACapCommand := MachineState.ActualState = WAITING_TAKE_A_CAP_COMMAND;
	gPusher.Feedbacks.CapReady := gPusher.Interface.Inputs.CapAtPickPosition;
	gPusher.Feedbacks.InitPosition := gPusher.Interface.Inputs.PusherInBackwardPosition;
	gPusher.Feedbacks.InitDone := gPusher.Feedbacks.InitPosition AND gPusher.Commands.Automatic.Init;

END_ACTION

ACTION ResetOutputsAction:

    memset(ADR(gPusher.Interface.Outputs),0,SIZEOF(gPusher.Interface.Outputs));

END_ACTION

ACTION ResetFeedbacksAction:

    memset(ADR(gPusher.Feedbacks),0,SIZEOF(gPusher.Feedbacks));

END_ACTION

ACTION MachineStateManagementAction:

    // Machine state timeout check
    MachineState.TimeoutTimer(IN := MachineState.TimeoutTimer.PT <> T#0S AND NOT MachineState.NewTriggerState);

    // Machine state change state logic
    MachineState.NewTriggerState := (MachineState.ActualState <> MachineState.NextState);
    IF MachineState.NewTriggerState THEN
        MachineState.OldState := MachineState.ActualState;
    END_IF
    MachineState.ActualState := MachineState.NextState;

END_ACTION

ACTION SetAlarmsAction:
	IF gPusher.Commands.Reset THEN
		Internal.Error := FALSE;
	END_IF

    // Timeouts alarms
	IF MachineState.TimeoutTimer.Q THEN
		CASE MachineState.ActualState OF
			MOVE_BACKWARD: MpAlarmXSet(gAlarmXCoreMpLink,'PusherTimeoutBackward'); // Edge alarm!
			MOVE_FORWARD: MpAlarmXSet(gAlarmXCoreMpLink,'PusherTimeoutForward'); // Edge alarm!
			WAITING_MAGAZINE: MpAlarmXSet(gAlarmXCoreMpLink,'PusherTimeoutMagazineEmpty'); // Edge alarm!
		END_CASE
		Internal.Error := TRUE;
		MachineState.NextState := ERROR;
	END_IF

	// PusherInvalidSensorsCombination
	IF gPusher.Interface.Inputs.PusherInBackwardPosition AND gPusher.Interface.Inputs.PusherInForwardPosition THEN
		MpAlarmXSet(gAlarmXCoreMpLink,'PusherInvalidSensorsCombination'); // Periodic alarm!
		Internal.Error := TRUE;
		MachineState.NextState := ERROR;
	ELSE
		MpAlarmXReset(gAlarmXCoreMpLink,'PusherInvalidSensorsCombination');
	END_IF

END_ACTION

ACTION ResetAlarmsAction:

	MpAlarmXReset(gAlarmXCoreMpLink,'PusherInvalidSensorsCombination');

END_ACTION
```

### PickerGlobalTypes.typ
```iecst
TYPE
	PickerType : 	STRUCT  (*Picker Main type*)
		Commands : PickerCommadsType;
		Feedbacks : PickerFeedbacksType;
		Interface : PickerInterfaceType;
	END_STRUCT;
	PickerCommadsType : 	STRUCT  (*Picker Commands type*)
		Enable : BOOL;
		Reset : BOOL;
		Manual : PickerManualCommadsType;
		Automatic : PickerAutomaticCommadsType;
	END_STRUCT;
	PickerFeedbacksType : 	STRUCT  (*Picker Feedbacks type*)
		Enabled : BOOL;
		WaitingPickCommand : BOOL;
		Error : BOOL;
		WaitingStart : BOOL;
		PickACapDone : BOOL;
		InitDone : BOOL;
		InitPosition : BOOL;
	END_STRUCT;
	PickerInterfaceType : 	STRUCT  (*Picker Interface type*)
		Inputs : PickerInterfaceInputsType;
		Outputs : PickerInterfaceOutputsType;
	END_STRUCT;
	PickerInterfaceOutputsType : 	STRUCT  (*Picker Interface Output type*)
		ArmForward : BOOL;
		ArmBackward : BOOL;
		GripperPick : BOOL;
	END_STRUCT;
	PickerInterfaceInputsType : 	STRUCT  (*Picker Interface Input type*)
		ArmBackward : BOOL;
		ArmForward : BOOL;
		GripperVacuum : BOOL;
	END_STRUCT;
	PickerAutomaticCommadsType : 	STRUCT  (*Picker Commands type*)
		PickACap : BOOL;
		Init : BOOL;
		Start : BOOL;
	END_STRUCT;
	PickerManualCommadsType : 	STRUCT  (*Picker Commands type*)
		Enable : BOOL;
		MoveForward : BOOL;
		MoveBackward : BOOL;
		ActivateGrip : BOOL;
	END_STRUCT;
END_TYPE
```

### PickerGlobalVariables.var
```iecst
VAR
    gPicker : PickerType;
END_VAR
```

### Program Logical/Source/Picker/PickerProgram (IEC)

#### Main.st - Init, cyclic, exit code
```iecst
//******************************************************************************************************
// Program: 	PickerProgram
// Author: 		Andrea Pennisi
// Rev.: 		1.0.0
// Date:		5.12.2023
//
// Description:
// This module is used to pick a cap from the pusher station to the conveyor.
// Only pneumatic motion in this module
//******************************************************************************************************

PROGRAM _INIT

    ResetOutputsAction;
    ResetFeedbacksAction;

    MachineState.NextState := WAITING_INIT;

END_PROGRAM

PROGRAM _CYCLIC
    // Enable module
    IF NOT gPicker.Commands.Enable THEN
        ResetOutputsAction;
		ResetFeedbacksAction;
		ResetAlarmsAction;
        RETURN;
    END_IF

	IF EDGENEG(gPicker.Commands.Automatic.Start) THEN
		IF MachineState.NextState <> ERROR THEN
			MachineState.NextState := WAITING_START;
		END_IF
	END_IF

	IF EDGEPOS(gPicker.Commands.Automatic.Init) THEN
		IF MachineState.NextState <> ERROR THEN
			MachineState.NextState := WAITING_INIT;
		END_IF
	END_IF

	// Alarms
	SetAlarmsAction;

    // Machine state
    MachineStateManagementAction;
    CASE MachineState.ActualState OF

		WAITING_INIT:
			MachineState.TimeoutTimer.PT := T#0S; // Timeout disabled in this state
			IF MachineState.NewTriggerState THEN
				ResetOutputsAction;
				gPicker.Feedbacks.PickACapDone := FALSE;
			END_IF

			IF gPicker.Commands.Automatic.Init THEN
				MachineState.NextState := MOVE_BACKWARD;

			ELSIF gPicker.Commands.Manual.Enable THEN
				MachineState.NextState := MANUALS;

			END_IF

		MANUALS:
			MachineState.TimeoutTimer.PT := T#0S; // Timeout disabled in this state
			// Manual commands
			gPicker.Interface.Outputs.ArmForward := gPicker.Commands.Manual.MoveForward;
			gPicker.Interface.Outputs.ArmBackward := gPicker.Commands.Manual.MoveBackward;
			gPicker.Interface.Outputs.GripperPick := gPicker.Commands.Manual.ActivateGrip;

			IF NOT gPicker.Commands.Manual.Enable THEN
				MachineState.NextState := WAITING_INIT;
			END_IF

		MOVE_BACKWARD:
			MachineState.TimeoutTimer.PT := T#3S;
			gPicker.Interface.Outputs.ArmBackward := TRUE;
			IF gPicker.Interface.Inputs.ArmBackward THEN
				gPicker.Interface.Outputs.ArmBackward := FALSE;
				MachineState.NextState := PLACE_CAP;
			END_IF

		PLACE_CAP:
			MachineState.TimeoutTimer.PT := T#3S;
			gPicker.Interface.Outputs.GripperPick := FALSE;
			IF NOT gPicker.Interface.Inputs.GripperVacuum THEN
				gPicker.Feedbacks.PickACapDone := Internal.CapPicked;
				Internal.CapPicked := FALSE;
				MachineState.NextState := WAITING_START;
			END_IF

		WAITING_START:
			MachineState.TimeoutTimer.PT := T#0S; // Timeout disabled in this state
			gPicker.Feedbacks.PickACapDone := FALSE;

			IF gPicker.Commands.Automatic.Start THEN
				MachineState.NextState := WAITING_PICK_COMMAND;

			ELSIF gPicker.Commands.Manual.Enable THEN
				MachineState.NextState := MANUALS;
			END_IF

        WAITING_PICK_COMMAND:
			MachineState.TimeoutTimer.PT := T#0S; // Timeout disabled in this state

			IF gPicker.Commands.Automatic.PickACap THEN
				gPicker.Feedbacks.PickACapDone := FALSE;
                MachineState.NextState := MOVE_FORWARD;
            END_IF

		MOVE_FORWARD:
			MachineState.TimeoutTimer.PT := T#3S;
			gPicker.Interface.Outputs.ArmForward := TRUE;
			IF gPicker.Interface.Inputs.ArmForward THEN
				gPicker.Interface.Outputs.ArmForward := FALSE;
				MachineState.NextState := PICK_CAP;
			END_IF

		PICK_CAP:
			MachineState.TimeoutTimer.PT := T#3S;
			gPicker.Interface.Outputs.GripperPick := TRUE;
			IF gPicker.Interface.Inputs.GripperVacuum THEN
				Internal.CapPicked := TRUE;
				MachineState.NextState := MOVE_BACKWARD;
			END_IF

        ERROR:
            MachineState.TimeoutTimer.PT := T#0S; // Timeout disabled in this state
			ResetOutputsAction;
			IF NOT Internal.Error THEN
				MachineState.NextState := WAITING_INIT;
			END_IF

        ELSE
            MachineState.NextState := WAITING_INIT;

    END_CASE

    FeedbacksUpdateAction;

END_PROGRAM

PROGRAM _EXIT

END_PROGRAM
```

#### Types.typ - Local data types
```iecst
TYPE
	MachineStateType : 	STRUCT  (*Machine state main type*)
		OldState : MachineStateEnum; (*Actual state*)
		ActualState : MachineStateEnum; (*Actual state*)
		NextState : MachineStateEnum; (*Next state*)
		NewTriggerState : BOOL; (*Trigger state change*)
		TimeoutTimer : TON; (*State timeout*)
	END_STRUCT;
	MachineStateEnum :
		( (*Machine State enumeration*)
		WAITING_INIT,
		MANUALS,
		WAITING_START,
		MOVE_BACKWARD, (*INIT state*)
		PLACE_CAP, (*WAITING state*)
		WAITING_PICK_COMMAND, (*ERROR state*)
		MOVE_FORWARD,
		PICK_CAP,
		ERROR
		);
	InternalType : 	STRUCT
		CapPicked : BOOL;
		Error : BOOL;
	END_STRUCT;
END_TYPE
```

#### Variables.var - Local variables
```iecst
VAR
	MachineState : MachineStateType;
	Internal : InternalType;
END_VAR
```

#### Actions.st
```iecst
ACTION FeedbacksUpdateAction:

	gPicker.Feedbacks.Enabled := TRUE;
    gPicker.Feedbacks.WaitingPickCommand := MachineState.ActualState = WAITING_PICK_COMMAND;
    gPicker.Feedbacks.Error := MachineState.ActualState = ERROR;
	gPicker.Feedbacks.InitPosition := gPicker.Interface.Inputs.ArmBackward AND NOT gPicker.Interface.Inputs.GripperVacuum;
	gPicker.Feedbacks.InitDone := gPicker.Feedbacks.InitPosition AND gPicker.Commands.Automatic.Init;

END_ACTION

ACTION ResetOutputsAction:

    memset(ADR(gPicker.Interface.Outputs),0,SIZEOF(gPicker.Interface.Outputs));

END_ACTION

ACTION ResetFeedbacksAction:

    memset(ADR(gPicker.Feedbacks),0,SIZEOF(gPicker.Feedbacks));

END_ACTION

ACTION MachineStateManagementAction:

    // Machine state timeout check
    MachineState.TimeoutTimer(IN := MachineState.TimeoutTimer.PT <> T#0S AND NOT MachineState.NewTriggerState);

	// Machine state change state logic
	MachineState.NewTriggerState := (MachineState.ActualState <> MachineState.NextState);
	IF MachineState.NewTriggerState THEN
		MachineState.OldState := MachineState.ActualState;
	END_IF
	MachineState.ActualState := MachineState.NextState;

END_ACTION

ACTION SetAlarmsAction:

	IF gPicker.Commands.Reset THEN
		Internal.Error := FALSE;
	END_IF

	// Timeouts alarms
	IF MachineState.TimeoutTimer.Q THEN
		CASE MachineState.ActualState OF
			MOVE_BACKWARD: MpAlarmXSet(gAlarmXCoreMpLink,'PickerTimeoutBackward'); // Edge alarm!
			MOVE_FORWARD: MpAlarmXSet(gAlarmXCoreMpLink,'PickerTimeoutForward'); // Edge alarm!
			PLACE_CAP: MpAlarmXSet(gAlarmXCoreMpLink,'PickerTimeoutVacuumPlace'); // Edge alarm!
			PICK_CAP: MpAlarmXSet(gAlarmXCoreMpLink,'PickerTimeoutVacuumPick'); // Edge alarm!
		END_CASE
		Internal.Error := TRUE;
		MachineState.NextState := ERROR;
	END_IF

	// PickupArmInvalidSensorsCombination
	IF gPicker.Interface.Inputs.ArmBackward AND gPicker.Interface.Inputs.ArmForward THEN
		MpAlarmXSet(gAlarmXCoreMpLink,'PickerInvalidSensorsCombination'); // Periodic alarm!
		Internal.Error := TRUE;
		MachineState.NextState := ERROR;
	ELSE
		MpAlarmXReset(gAlarmXCoreMpLink,'PickerInvalidSensorsCombination');
	END_IF

END_ACTION

ACTION ResetAlarmsAction:

	MpAlarmXReset(gAlarmXCoreMpLink,'PickerInvalidSensorsCombination');

END_ACTION
```

### ConveyorGlobalTypes.typ
```iecst
TYPE
	ConveyorType : 	STRUCT  (*Conveyor Main type*)
		Commands : ConveyorCommadsType;
		Feedbacks : ConveyorFeedbacksType;
		Parameters : ConveyorParametersType;
		Interface : ConveyorInterfaceType;
	END_STRUCT;
	ConveyorCommadsType : 	STRUCT  (*Conveyor Commands type*)
		Enable : BOOL;
		Reset : BOOL;
		Automatic : ConveyorAutomaticCommadsType;
		Manual : ConveyorManualCommadsType;
	END_STRUCT;
	ConveyorFeedbacksType : 	STRUCT  (*Conveyor Feedbacks type*)
		Enabled : BOOL;
		WaitingStart : BOOL;
		Error : BOOL;
		WaitingCap : BOOL;
		DeliverCapDone : BOOL;
		InitDone : BOOL;
		AxisHomed : BOOL;
		AxisPowered : BOOL;
		InitPosition : BOOL;
		AxisSpeed : REAL;
		AxisPosition : LREAL;
		CapsOnConveyor : USINT;
	END_STRUCT;
	ConveyorParametersType : 	STRUCT  (*Conveyor Parameters type*)
		TargetSpeed : REAL := 50;
		Acceleration : REAL := 5000;
	END_STRUCT;
	ConveyorInterfaceType : 	STRUCT  (*Conveyor Interface type*)
		Inputs : ConveyorInterfaceInputsType;
		Outputs : ConveyorInterfaceOutputsType;
	END_STRUCT;
	ConveyorInterfaceOutputsType : 	STRUCT  (*Conveyor Interface Output type*)
		SetSpeed : REAL;
	END_STRUCT;
	ConveyorInterfaceInputsType : 	STRUCT  (*Conveyor Interface Input type*)
		CapInStartPosition : BOOL;
		CapInExitPosition : BOOL;
	END_STRUCT;
	ConveyorAutomaticCommadsType : 	STRUCT  (*Conveyor Commands type*)
		Start : BOOL;
		Init : BOOL;
		DeliverCap : BOOL;
	END_STRUCT;
	ConveyorManualCommadsType : 	STRUCT  (*Conveyor Commands type*)
		Enable : BOOL;
		PowerOn : BOOL;
		Move : BOOL;
		Home : BOOL;
		Speed : REAL := 50;
	END_STRUCT;
END_TYPE
```

### ConveyorGlobalVariables.var
```iecst
VAR
    gConveyor : ConveyorType;
END_VAR
```

### Program Logical/Source/Conveyor/ConveyorProgram (IEC)

#### Main.st - Init, cyclic, exit code
```iecst
//******************************************************************************************************
// Program: 	ConveyorProgram
// Author: 		Andrea Pennisi
// Rev.: 		1.0.0
// Date:		5.12.2023
//
// Description:
// This module is used to deliver the cap from the starting position of the conveyor to the exit.
// An axis is controlled by mappMotion tools. The control is made in velocity.
//******************************************************************************************************

PROGRAM _INIT

    ResetOutputsAction;
    ResetFeedbacksAction;

	Internal.Parameters.Homing.Mode := mcHOMING_ABSOLUTE;

    MachineState.NextState := WAITING_INIT;

END_PROGRAM

PROGRAM _CYCLIC

	MotionAction;

    // Enable module
    IF NOT gConveyor.Commands.Enable THEN
        ResetOutputsAction;
		ResetFeedbacksAction;
		ResetAlarmsAction;
		ResetMotionCommands;
        RETURN;
    END_IF

	IF EDGENEG(gConveyor.Commands.Automatic.Start) THEN
		IF MachineState.NextState <> ERROR THEN
			MachineState.NextState := WAITING_START;
		END_IF
	END_IF

	IF EDGEPOS(gConveyor.Commands.Automatic.Init) THEN
		IF MachineState.NextState <> ERROR THEN
			MachineState.NextState := WAITING_INIT;
		END_IF
	END_IF

	// Alarms
	SetAlarmsAction;

    // Machine state
    MachineStateManagementAction;
    CASE MachineState.ActualState OF

		WAITING_INIT:
			MachineState.TimeoutTimer.PT := T#0S; // Timeout disabled in this state
			IF MachineState.NewTriggerState THEN
				ResetOutputsAction;
				ResetMotionCommands;
			END_IF

			IF gConveyor.Commands.Automatic.Init THEN
				gConveyor.Feedbacks.CapsOnConveyor := 0;
				MachineState.NextState := HOMING;

			ELSIF gConveyor.Commands.Manual.Enable THEN
				MachineState.NextState := MANUALS;

			END_IF

		MANUALS:
			MachineState.TimeoutTimer.PT := T#0S; // Timeout disabled in this state

			Internal.Parameters.Velocity := gConveyor.Commands.Manual.Speed;
			IF Internal.Parameters.Velocity>0 THEN
				Internal.Parameters.Direction := mcDIR_POSITIVE;
			ELSE
				Internal.Parameters.Direction := mcDIR_NEGATIVE;
			END_IF

			Internal.Axis.Home := gConveyor.Commands.Manual.Home AND Internal.Axis.Active AND NOT Internal.Axis.Error;
			IF Internal.Axis.IsHomed THEN
				Internal.Axis.Power := gConveyor.Commands.Manual.PowerOn AND Internal.Axis.Active AND NOT Internal.Axis.Error;
				IF Internal.Axis.PowerOn THEN
					Internal.Axis.MoveVelocity := gConveyor.Commands.Manual.Move AND Internal.Axis.Active AND NOT Internal.Axis.Error;
				ELSE
					Internal.Axis.MoveVelocity := FALSE;
				END_IF
			ELSE
				Internal.Axis.Power := FALSE;
				Internal.Axis.MoveVelocity := FALSE;
			END_IF

			IF NOT gConveyor.Commands.Manual.Enable THEN
				MachineState.NextState := WAITING_INIT;
			END_IF

		HOMING:
			MachineState.TimeoutTimer.PT := T#3S;
			IF Internal.Axis.IsHomed THEN
				Internal.Axis.Home := FALSE;
				MachineState.NextState := POWER_ON;
			ELSE
				Internal.Axis.Home := Internal.Axis.Active AND NOT Internal.Axis.Error;
			END_IF

		POWER_ON:
			MachineState.TimeoutTimer.PT := T#3S;
			Internal.Axis.Power := Internal.Axis.Active AND NOT Internal.Axis.Error;
			IF Internal.Axis.PowerOn THEN
				IF gConveyor.Commands.Automatic.Init THEN
					MachineState.NextState := INIT;
				ELSE
					MachineState.NextState := WAITING_CAP;
				END_IF
			END_IF

		INIT:
			MachineState.TimeoutTimer.PT := T#30S;
			IF MachineState.NewTriggerState THEN
				Internal.Parameters.Velocity := gConveyor.Parameters.TargetSpeed;
				Internal.Parameters.Direction := mcDIR_POSITIVE;
			END_IF
			Internal.Axis.MoveAbsolute := Internal.Axis.Active AND NOT Internal.Axis.Error;
			IF Internal.Axis.MoveDone THEN
				Internal.Axis.MoveAbsolute := FALSE;
				MachineState.NextState := WAITING_START;
			END_IF

        WAITING_START:
			MachineState.TimeoutTimer.PT := T#0S; // Timeout disabled in this state
			IF MachineState.NewTriggerState THEN
				Internal.Axis.Power := FALSE;
			END_IF
			gConveyor.Feedbacks.DeliverCapDone := FALSE;
            IF gConveyor.Commands.Automatic.Start THEN
				MachineState.NextState := POWER_ON;

			ELSIF gConveyor.Commands.Manual.Enable THEN
				MachineState.NextState := MANUALS;
            END_IF

		WAITING_CAP:
			MachineState.TimeoutTimer.PT := T#0S; // Timeout disabled in this state
			IF gConveyor.Interface.Inputs.CapInStartPosition AND gConveyor.Commands.Automatic.DeliverCap THEN
				gConveyor.Feedbacks.DeliverCapDone := FALSE;
				MachineState.NextState := MOTION;
			END_IF

		MOTION:
			MachineState.TimeoutTimer.PT := T#30S;
			IF MachineState.NewTriggerState THEN
				Internal.Parameters.Direction := mcDIR_POSITIVE;
			END_IF

			// On-fly velocity change
			IF Internal.Parameters.Velocity <> gConveyor.Parameters.TargetSpeed THEN
				Internal.Parameters.Velocity := gConveyor.Parameters.TargetSpeed;
				Internal.Axis.Update := TRUE;
			ELSIF Internal.Axis.UpdateDone THEN
				Internal.Axis.Update := FALSE;
			END_IF

			Internal.Axis.MoveVelocity := TRUE;
			IF EDGENEG(gConveyor.Interface.Inputs.CapInExitPosition) THEN
				gConveyor.Feedbacks.DeliverCapDone := TRUE;
				Internal.Axis.MoveVelocity := FALSE;
				Internal.Axis.Update := FALSE;
				MachineState.NextState := WAITING_CAP;
			END_IF

        ERROR:
            MachineState.TimeoutTimer.PT := T#0S; // Timeout disabled in this state
			ResetOutputsAction;
			ResetMotionCommands;
			IF NOT Internal.Error THEN
				MachineState.NextState := WAITING_INIT;
			END_IF

        ELSE
            MachineState.NextState := WAITING_START;

    END_CASE

    FeedbacksUpdateAction;

END_PROGRAM

PROGRAM _EXIT

END_PROGRAM
```

#### Types.typ - Local data types
```iecst
TYPE
	MachineStateType : 	STRUCT  (*Machine state main type*)
		OldState : MachineStateEnum; (*Actual state*)
		ActualState : MachineStateEnum; (*Actual state*)
		NextState : MachineStateEnum; (*Next state*)
		NewTriggerState : BOOL; (*Trigger state change*)
		TimeoutTimer : TON; (*State timeout*)
	END_STRUCT;
	MachineStateEnum :
		( (*Machine State enumeration*)
		WAITING_INIT, (*WAITING state*)
		MANUALS,
		WAITING_START,
		HOMING,
		POWER_ON,
		INIT,
		WAITING_CAP,
		MOTION,
		ERROR (*ERROR state*)
		);
	InternalType : 	STRUCT
		Axis : MpAxisBasic;
		Parameters : MpAxisBasicParType;
		Error : BOOL;
	END_STRUCT;
END_TYPE
```

#### Variables.var - Local variables
```iecst
VAR
	MachineState : MachineStateType;
	Internal : InternalType;
END_VAR
```

#### Actions.st
```iecst
ACTION FeedbacksUpdateAction:

    gConveyor.Feedbacks.Enabled := TRUE;
    gConveyor.Feedbacks.WaitingStart := MachineState.ActualState = WAITING_START;
    gConveyor.Feedbacks.Error := MachineState.ActualState = ERROR;
	gConveyor.Feedbacks.WaitingCap := MachineState.ActualState = WAITING_CAP;
	gConveyor.Feedbacks.AxisHomed := Internal.Axis.IsHomed;
	gConveyor.Feedbacks.AxisPowered := Internal.Axis.PowerOn;
	gConveyor.Feedbacks.InitPosition := ABS(Internal.Axis.Position - Internal.Parameters.Position)<0.1;
	gConveyor.Feedbacks.InitDone := gConveyor.Feedbacks.InitPosition AND gConveyor.Commands.Automatic.Init;
	gConveyor.Feedbacks.AxisSpeed := Internal.Axis.Velocity;
	gConveyor.Feedbacks.AxisPosition := Internal.Axis.Position;

	IF EDGEPOS(gConveyor.Interface.Inputs.CapInStartPosition) AND gConveyor.Commands.Automatic.Start THEN
		gConveyor.Feedbacks.CapsOnConveyor := gConveyor.Feedbacks.CapsOnConveyor + 1;

	ELSIF gConveyor.Interface.Inputs.CapInStartPosition AND gConveyor.Commands.Automatic.Start AND gConveyor.Feedbacks.CapsOnConveyor = 0 THEN
		gConveyor.Feedbacks.CapsOnConveyor := gConveyor.Feedbacks.CapsOnConveyor + 1;
	END_IF

	IF EDGEPOS(gConveyor.Interface.Inputs.CapInExitPosition) THEN
		IF gConveyor.Feedbacks.CapsOnConveyor>1 THEN
			gConveyor.Feedbacks.CapsOnConveyor := gConveyor.Feedbacks.CapsOnConveyor - 1;
		ELSE
			gConveyor.Feedbacks.CapsOnConveyor := 0;
		END_IF
	END_IF

END_ACTION

ACTION ResetOutputsAction:

	memset(ADR(gConveyor.Interface.Outputs),0,SIZEOF(gConveyor.Interface.Outputs));

END_ACTION

ACTION ResetMotionCommands:
	Internal.Axis.Power := FALSE;
	Internal.Axis.Home := FALSE;
	Internal.Axis.MoveVelocity := FALSE;
	Internal.Axis.MoveAbsolute := FALSE;
	Internal.Axis.Update := FALSE;
END_ACTION

ACTION ResetFeedbacksAction:

    memset(ADR(gConveyor.Feedbacks),0,SIZEOF(gConveyor.Feedbacks));

END_ACTION

ACTION MachineStateManagementAction:

    // Machine state timeout check
    MachineState.TimeoutTimer(IN := MachineState.TimeoutTimer.PT <> T#0S AND NOT MachineState.NewTriggerState);

    // Machine state change state logic
    MachineState.NewTriggerState := (MachineState.ActualState <> MachineState.NextState);
    IF MachineState.NewTriggerState THEN
        MachineState.OldState := MachineState.ActualState;
    END_IF
    MachineState.ActualState := MachineState.NextState;

END_ACTION

ACTION SetAlarmsAction:

	IF gConveyor.Commands.Reset THEN
		Internal.Error := FALSE;
	END_IF

	// Timeouts
	IF MachineState.TimeoutTimer.Q THEN

		CASE MachineState.ActualState OF
			HOMING: MpAlarmXSet(gAlarmXCoreMpLink,'ConveyorTimeoutHoming'); // Edge alarm!
			POWER_ON: MpAlarmXSet(gAlarmXCoreMpLink,'ConveyorTimeoutPowerOn'); // Edge alarm!
			MOTION: MpAlarmXSet(gAlarmXCoreMpLink,'ConveyorMissedCap'); // Edge alarm!
			INIT: MpAlarmXSet(gAlarmXCoreMpLink,'ConveyorInitFail'); // Edge alarm!
		END_CASE

		Internal.Error := TRUE;
		MachineState.NextState := ERROR;
	END_IF

	// ConveyorAxisError
	IF Internal.Axis.Error THEN
		MpAlarmXSet(gAlarmXCoreMpLink,'ConveyorAxisError');
		Internal.Error := TRUE;
		MachineState.NextState := ERROR;
	ELSE
		MpAlarmXReset(gAlarmXCoreMpLink,'ConveyorAxisError');
	END_IF

	// ConveyorTooManyCaps
	IF gConveyor.Commands.Reset THEN
		gConveyor.Feedbacks.CapsOnConveyor := 0;
	END_IF
	IF gConveyor.Feedbacks.CapsOnConveyor > 1 THEN
		MpAlarmXSet(gAlarmXCoreMpLink,'ConveyorTooManyCaps');
		Internal.Error := TRUE;
		MachineState.NextState := ERROR;
	ELSE
		MpAlarmXReset(gAlarmXCoreMpLink,'ConveyorTooManyCaps');
	END_IF
END_ACTION

ACTION ResetAlarmsAction:

	MpAlarmXReset(gAlarmXCoreMpLink,'ConveyorAxisError');

END_ACTION
```

#### MotionAction.ld
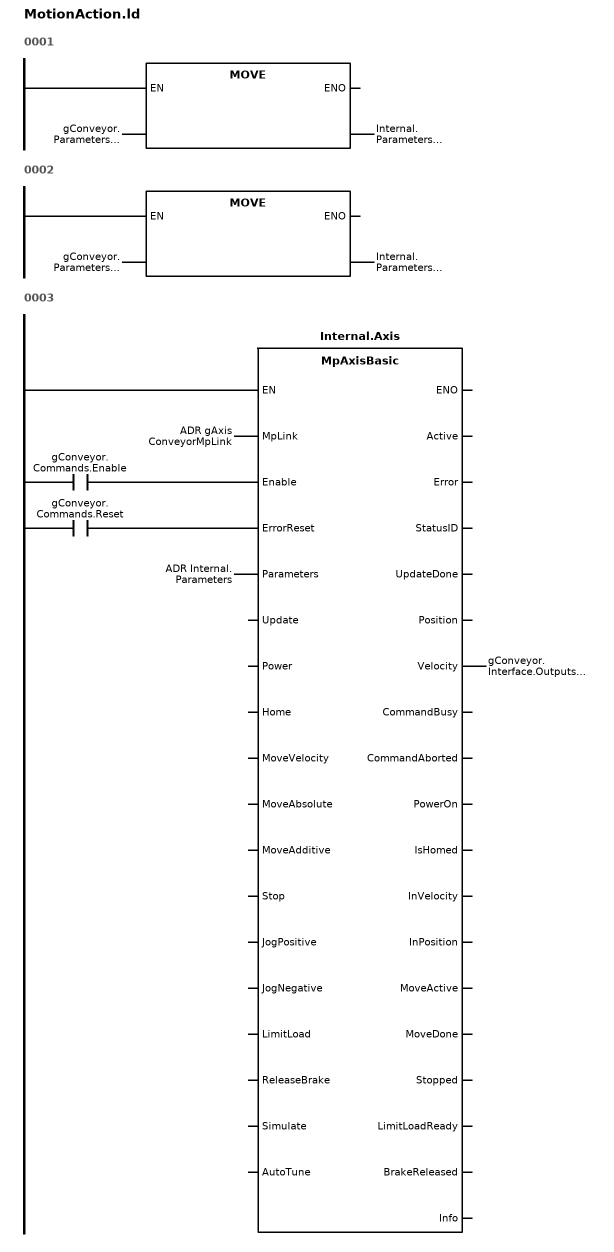
Ladder, written as Structured Text:
```iecst
ACTION MotionAction:
(* Network 1 *)
Internal.Parameters.Deceleration := gConveyor.Parameters.Acceleration;

(* Network 2 *)
Internal.Parameters.Acceleration := gConveyor.Parameters.Acceleration;

(* Network 3 *)
Internal.Axis(MpLink := ADR(gAxisConveyorMpLink), Enable := gConveyor.Commands.Enable, ErrorReset := gConveyor.Commands.Reset, Parameters := ADR(Internal.Parameters));
gConveyor.Interface.Outputs.SetSpeed := Internal.Axis.Velocity;
END_ACTION
```

### StamperGlobalTypes.typ
```iecst
TYPE
	StamperType : 	STRUCT  (*Stamper Main type*)
		Commands : StamperCommadsType;
		Feedbacks : StamperFeedbacksType;
		Parameters : StamperParametersType;
		Interface : StamperInterfaceType;
	END_STRUCT;
	StamperCommadsType : 	STRUCT  (*Stamper Commands type*)
		Enable : BOOL;
		Reset : BOOL;
		Automatic : StamperAutomaticCommadsType;
		Manual : StamperManualCommadsType;
	END_STRUCT;
	StamperFeedbacksType : 	STRUCT  (*Stamper Feedbacks type*)
		Enabled : BOOL;
		WaitingStart : BOOL;
		Error : BOOL;
		OnSyncMotion : BOOL;
		WaitingCap : BOOL;
		StampCapDone : BOOL;
		InitDone : BOOL;
		InitPosition : BOOL;
		AxisSpeed : REAL;
		AxisPosition : LREAL;
		AxisHomed : BOOL;
		AxisPowered : BOOL;
	END_STRUCT;
	StamperParametersType : 	STRUCT  (*Stamper Parameters type*)
		Offset : REAL := 65;
		Speed : REAL := 10000;
		Acceleration : REAL := 20000;
	END_STRUCT;
	StamperInterfaceType : 	STRUCT  (*Stamper Interface type*)
		Inputs : StamperInterfaceInputsType;
		Outputs : StamperInterfaceOutputsType;
	END_STRUCT;
	StamperInterfaceOutputsType : 	STRUCT  (*Stamper Interface Output type*)
		StampForward : BOOL;
		SetPosition : LREAL;
	END_STRUCT;
	StamperInterfaceInputsType : 	STRUCT  (*Stamper Interface Input type*)
		ActualPosition : REAL;
		StampIsForward : BOOL;
		StampIsBackward : BOOL;
	END_STRUCT;
	StamperAutomaticCommadsType : 	STRUCT  (*Stamper Commands type*)
		Start : BOOL;
		Init : BOOL;
		StampCap : BOOL;
	END_STRUCT;
	StamperManualCommadsType : 	STRUCT  (*Stamper Commands type*)
		Enable : BOOL;
		StamperForward : BOOL;
		Position : LREAL;
		Speed : REAL := 50;
		PowerOn : BOOL;
		Move : BOOL;
		Home : BOOL;
	END_STRUCT;
END_TYPE
```

### StamperGlobalVariables.var
```iecst
VAR
    gStamper : StamperType;
END_VAR
```

### Program Logical/Source/Stamper/StamperProgram (IEC)

#### Main.st - Init, cyclic, exit code
```iecst
//******************************************************************************************************
// Program: 	StamperProgram
// Author: 		Andrea Pennisi
// Rev.: 		1.0.0
// Date:		5.12.2023
//
// Description:
// This module is used to stamp the logo in the cap.
// An axis is controlled by mappMotion tools. The control is made by a cam linked to the Conveyor module axis.
//******************************************************************************************************
PROGRAM _INIT

    ResetOutputsAction;
    ResetFeedbacksAction;

	Internal.Parameters.Homing.Mode := mcHOMING_DIRECT;

	Internal.Offset.AdvancedParameters.ShiftMode := mcSHIFT_ABSOLUTE;
	Internal.Offset.Enable := TRUE;

    MachineState.NextState := WAITING_INIT;

END_PROGRAM

PROGRAM _CYCLIC

	MotionAction;

    // Enable module
    IF NOT gStamper.Commands.Enable THEN
        ResetOutputsAction;
		ResetFeedbacksAction;
		ResetAlarmsAction;
		ResetMotionCommands;
        RETURN;
    END_IF

	IF EDGENEG(gStamper.Commands.Automatic.Start) THEN
		IF MachineState.NextState <> ERROR THEN
			MachineState.NextState := WAITING_START;
		END_IF
	END_IF

	IF EDGEPOS(gStamper.Commands.Automatic.Init) THEN
		IF MachineState.NextState <> ERROR THEN
			MachineState.NextState := WAITING_INIT;
		END_IF
	END_IF

	// Alarms
	SetAlarmsAction;

    // Machine state
    MachineStateManagementAction;
    CASE MachineState.ActualState OF

		WAITING_INIT:
			MachineState.TimeoutTimer.PT := T#0S; // Timeout disabled in this state
			IF MachineState.NewTriggerState THEN
				ResetOutputsAction;
				ResetMotionCommands;
				Internal.CamStartTrigger := FALSE;
			END_IF

			IF gStamper.Commands.Automatic.Init THEN
				MachineState.NextState := HOMING;

			ELSIF gStamper.Commands.Manual.Enable THEN
				MachineState.NextState := MANUAL;

			END_IF

		MANUAL:
			MachineState.TimeoutTimer.PT := T#0S; // Timeout disabled in this state

			Internal.Parameters.Velocity := gStamper.Commands.Manual.Speed;
			Internal.Parameters.Position := gStamper.Commands.Manual.Position;

			gStamper.Interface.Outputs.StampForward := gStamper.Commands.Manual.StamperForward;

			Internal.Axis.Home := gStamper.Commands.Manual.Home AND Internal.Axis.Active AND NOT Internal.Axis.Error;
			IF Internal.Axis.IsHomed THEN
				Internal.Axis.Power := gStamper.Commands.Manual.PowerOn AND Internal.Axis.Active AND NOT Internal.Axis.Error;
				IF Internal.Axis.PowerOn THEN
					Internal.Axis.MoveAbsolute := gStamper.Commands.Manual.Move AND Internal.Axis.Active AND NOT Internal.Axis.Error;
				ELSE
					Internal.Axis.MoveAbsolute := FALSE;
				END_IF
			ELSE
				Internal.Axis.Power := FALSE;
				Internal.Axis.MoveAbsolute := FALSE;
			END_IF

			IF NOT gStamper.Commands.Manual.Enable THEN
				MachineState.NextState := WAITING_INIT;
			END_IF

		HOMING:
			MachineState.TimeoutTimer.PT := T#3S;
			IF Internal.Axis.IsHomed THEN
				Internal.Axis.Home := FALSE;
				MachineState.NextState := POWER_ON;
			ELSE
				Internal.Axis.Home := Internal.Axis.Active AND NOT Internal.Axis.Error;
			END_IF

		POWER_ON:
			MachineState.TimeoutTimer.PT := T#3S;

			Internal.Axis.Power := Internal.Axis.Active AND NOT Internal.Axis.Error;
			IF Internal.Axis.PowerOn THEN
				IF gStamper.Commands.Automatic.Init THEN
					MachineState.NextState := INIT;
				ELSE
					MachineState.NextState := ACTIVATE_CAM;
				END_IF
			END_IF

		INIT:
			MachineState.TimeoutTimer.PT := T#15S;
			Internal.Parameters.Velocity := gStamper.Parameters.Speed;
			Internal.Parameters.Position := 0;
			Internal.Axis.MoveAbsolute := Internal.Axis.Active AND NOT Internal.Axis.Error;
			IF Internal.Axis.MoveDone THEN
				Internal.OffsetToDo := TRUE;
				Internal.Axis.MoveAbsolute := FALSE;
				MachineState.NextState := WAITING_START;
			END_IF

        WAITING_START:
			MachineState.TimeoutTimer.PT := T#0S; // Timeout disabled in this state
			IF MachineState.NewTriggerState THEN
				ResetMotionCommands;
				Internal.Parameters.Velocity := gStamper.Parameters.Speed;
			END_IF

			IF gStamper.Commands.Automatic.Start THEN
				gStamper.Feedbacks.StampCapDone := FALSE;
				MachineState.NextState := POWER_ON;

			ELSIF gStamper.Commands.Manual.Enable THEN
				MachineState.NextState := MANUAL;
            END_IF

		ACTIVATE_CAM:
			MachineState.TimeoutTimer.PT := T#0S; // Timeout disabled in this state
			Internal.Cam.Enable := TRUE;
			Internal.Cam.Start := TRUE;
			IF Internal.Axis.Info.PLCopenState = mcAXIS_SYNCHRONIZED_MOTION THEN
				MachineState.NextState := WAITING_CAP;
			END_IF

		WAITING_CAP:
			MachineState.TimeoutTimer.PT := T#0S; // Timeout disabled in this state
			IF gStamper.Commands.Automatic.StampCap THEN
				gStamper.Feedbacks.StampCapDone := FALSE;
				Internal.CamStartTrigger := TRUE;
			END_IF

			IF Internal.Cam.InCam AND Internal.Cam.ActualStateIndex = 1 THEN // Syncronized motion
				Internal.CamStartTrigger := FALSE;
				MachineState.NextState := STAMP_FORWARD;
			END_IF

		STAMP_FORWARD:
			MachineState.TimeoutTimer.PT := T#3S;

			gStamper.Interface.Outputs.StampForward := TRUE;
			IF gStamper.Interface.Inputs.StampIsForward THEN
				MachineState.NextState := STAMPING;
			END_IF

		STAMPING:
			MachineState.TimeoutTimer.PT := T#15S;

			IF Internal.Cam.ActualStateIndex <> 1 THEN
				gStamper.Interface.Outputs.StampForward := FALSE;
				MachineState.NextState := STAMP_BACKWARD;
			END_IF

		STAMP_BACKWARD:
			MachineState.TimeoutTimer.PT := T#3S;

			IF gStamper.Interface.Inputs.StampIsBackward THEN
				gStamper.Feedbacks.StampCapDone := TRUE;
				MachineState.NextState := WAITING_CAP;
			END_IF

        ERROR:
            MachineState.TimeoutTimer.PT := T#0S; // Timeout disabled in this state
			ResetOutputsAction;
			ResetMotionCommands;
			IF NOT Internal.Error THEN
				MachineState.NextState := WAITING_INIT;
			END_IF

        ELSE
            MachineState.NextState := WAITING_START;

    END_CASE

	OffsetManagement;

    FeedbacksUpdateAction;

END_PROGRAM

PROGRAM _EXIT

END_PROGRAM
```

#### Types.typ - Local data types
```iecst
TYPE
	MachineStateType : 	STRUCT  (*Machine state main type*)
		OldState : MachineStateEnum; (*Actual state*)
		ActualState : MachineStateEnum; (*Actual state*)
		NextState : MachineStateEnum; (*Next state*)
		NewTriggerState : BOOL; (*Trigger state change*)
		TimeoutTimer : TON; (*State timeout*)
	END_STRUCT;
	MachineStateEnum :
		( (*Machine State enumeration*)
		WAITING_INIT,
		MANUAL,
		WAITING_START, (*WAITING state*)
		HOMING,
		POWER_ON, (*INIT state*)
		INIT,
		ACTIVATE_CAM,
		WAITING_CAP,
		STAMP_FORWARD,
		STAMPING,
		STAMP_BACKWARD,
		ERROR (*ERROR state*)
		);
	InternalType : 	STRUCT
		Axis : MpAxisBasic;
		Parameters : MpAxisBasicParType;
		Cam : MC_BR_CamAutomatCommand;
		Offset : MC_BR_Offset;
		LastOffset : LREAL;
		CamStartTrigger : BOOL;
		Error : BOOL;
		OffsetToDo : BOOL;
	END_STRUCT;
END_TYPE
```

#### Variables.var - Local variables
```iecst
VAR
	MachineState : MachineStateType;
	Internal : InternalType;
END_VAR
```

#### Actions.st
```iecst
ACTION FeedbacksUpdateAction:

    gStamper.Feedbacks.Enabled := TRUE;
    gStamper.Feedbacks.WaitingStart := (MachineState.ActualState = WAITING_START);
	gStamper.Feedbacks.Error := (MachineState.ActualState = ERROR);
	gStamper.Feedbacks.OnSyncMotion := Internal.Cam.InCam;
	gStamper.Feedbacks.WaitingCap := (Internal.Cam.ActualStateIndex = 0) AND (MachineState.ActualState = WAITING_CAP);
	gStamper.Feedbacks.InitPosition := ABS(Internal.Axis.Position - Internal.Parameters.Position)<0.1;
	gStamper.Feedbacks.InitDone := gStamper.Feedbacks.InitPosition AND gStamper.Commands.Automatic.Init;
	gStamper.Feedbacks.AxisHomed := Internal.Axis.IsHomed;
	gStamper.Feedbacks.AxisPowered := Internal.Axis.PowerOn;
	gStamper.Feedbacks.AxisSpeed := Internal.Axis.Velocity;
	gStamper.Feedbacks.AxisPosition := Internal.Axis.Position;

END_ACTION

ACTION ResetOutputsAction:

    memset(ADR(gStamper.Interface.Outputs),0,SIZEOF(gStamper.Interface.Outputs));

END_ACTION

ACTION ResetFeedbacksAction:

    memset(ADR(gStamper.Feedbacks),0,SIZEOF(gStamper.Feedbacks));

END_ACTION

ACTION ResetMotionCommands:
	Internal.Axis.Power := FALSE;
	Internal.Axis.Home := FALSE;
	Internal.Axis.MoveVelocity := FALSE;
	Internal.Axis.MoveAbsolute := FALSE;

	Internal.Cam.Enable := FALSE;
	Internal.Cam.Start := FALSE;

	Internal.Offset.Enable := FALSE;
	Internal.Offset.StartShift := FALSE;
END_ACTION

ACTION MachineStateManagementAction:

    // Machine state timeout check
    MachineState.TimeoutTimer(IN := MachineState.TimeoutTimer.PT <> T#0S AND NOT MachineState.NewTriggerState);

    // Machine state change state logic
    MachineState.NewTriggerState := (MachineState.ActualState <> MachineState.NextState);
    IF MachineState.NewTriggerState THEN
        MachineState.OldState := MachineState.ActualState;
    END_IF
    MachineState.ActualState := MachineState.NextState;

END_ACTION

ACTION SetAlarmsAction:

	IF gStamper.Commands.Reset THEN
		Internal.Error := FALSE;
	END_IF

	IF MachineState.TimeoutTimer.Q THEN

		CASE MachineState.ActualState OF
			HOMING: MpAlarmXSet(gAlarmXCoreMpLink,'StamperTimeoutHoming'); // Edge alarm!
			POWER_ON: MpAlarmXSet(gAlarmXCoreMpLink,'StamperTimeoutPowerOn'); // Edge alarm!
			STAMP_FORWARD: MpAlarmXSet(gAlarmXCoreMpLink,'StamperTimeoutStampForward'); // Edge alarm!
			STAMP_BACKWARD: MpAlarmXSet(gAlarmXCoreMpLink,'StamperTimeoutStampBackward'); // Edge alarm!
			ACTIVATE_CAM: MpAlarmXSet(gAlarmXCoreMpLink,'StamperAxisTimeout'); // Edge alarm!
			STAMPING: MpAlarmXSet(gAlarmXCoreMpLink,'StamperAxisTimeout'); // Edge alarm!
		END_CASE

		Internal.Error := TRUE;
		MachineState.NextState := ERROR;
	END_IF

	IF Internal.Axis.Error OR Internal.Cam.Error OR Internal.Offset.Error THEN
		MpAlarmXSet(gAlarmXCoreMpLink,'StamperAxisError');
		Internal.Error := TRUE;
		MachineState.NextState := ERROR;
	ELSE
		MpAlarmXReset(gAlarmXCoreMpLink,'StamperAxisError');
	END_IF

	IF gStamper.Interface.Inputs.StampIsForward AND gStamper.Interface.Inputs.StampIsBackward THEN
		MpAlarmXSet(gAlarmXCoreMpLink,'StamperInvalidSensorsCombination');
		Internal.Error := TRUE;
		MachineState.NextState := ERROR;
	ELSE
		MpAlarmXReset(gAlarmXCoreMpLink,'StamperInvalidSensorsCombination');
	END_IF

END_ACTION

ACTION ResetAlarmsAction:

	MpAlarmXReset(gAlarmXCoreMpLink,'StamperInvalidSensorsCombination');

END_ACTION

ACTION OffsetManagement:

	Internal.Offset.Enable := Internal.Axis.Info.PLCopenState = mcAXIS_SYNCHRONIZED_MOTION;
	Internal.Offset.StartShift := (Internal.OffsetToDo OR Internal.LastOffset <> gStamper.Parameters.Offset) AND Internal.Offset.Valid;
	Internal.LastOffset := gStamper.Parameters.Offset;
	IF Internal.OffsetToDo AND Internal.Offset.StartShift THEN
		Internal.OffsetToDo := FALSE;
	END_IF

END_ACTION
```

#### MotionAction.ld
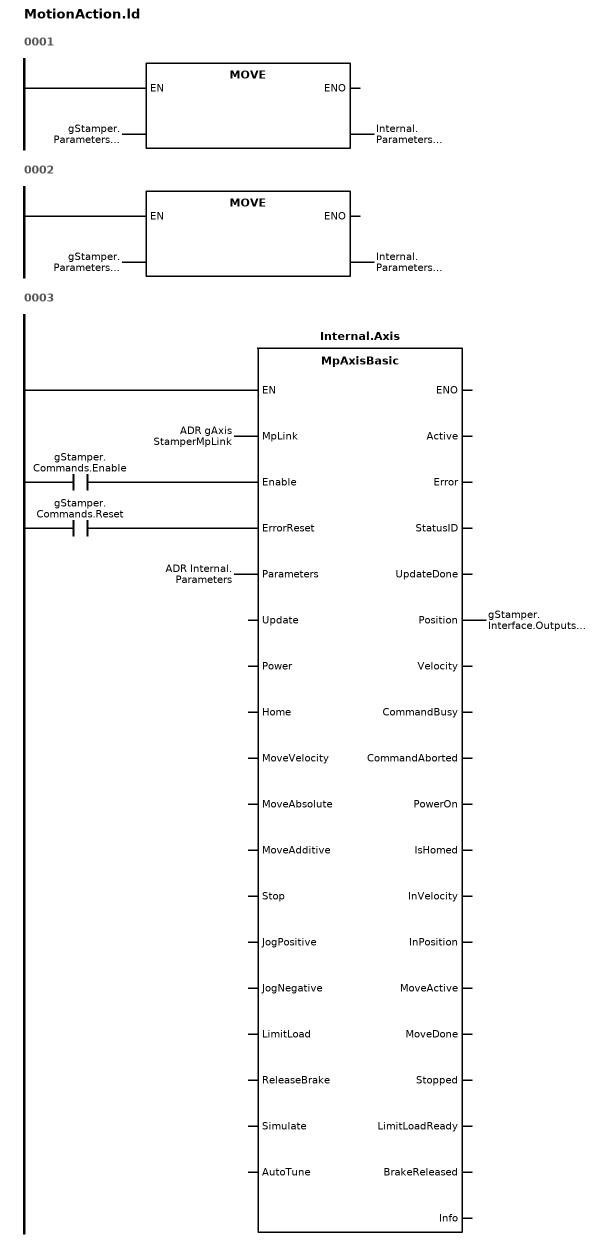
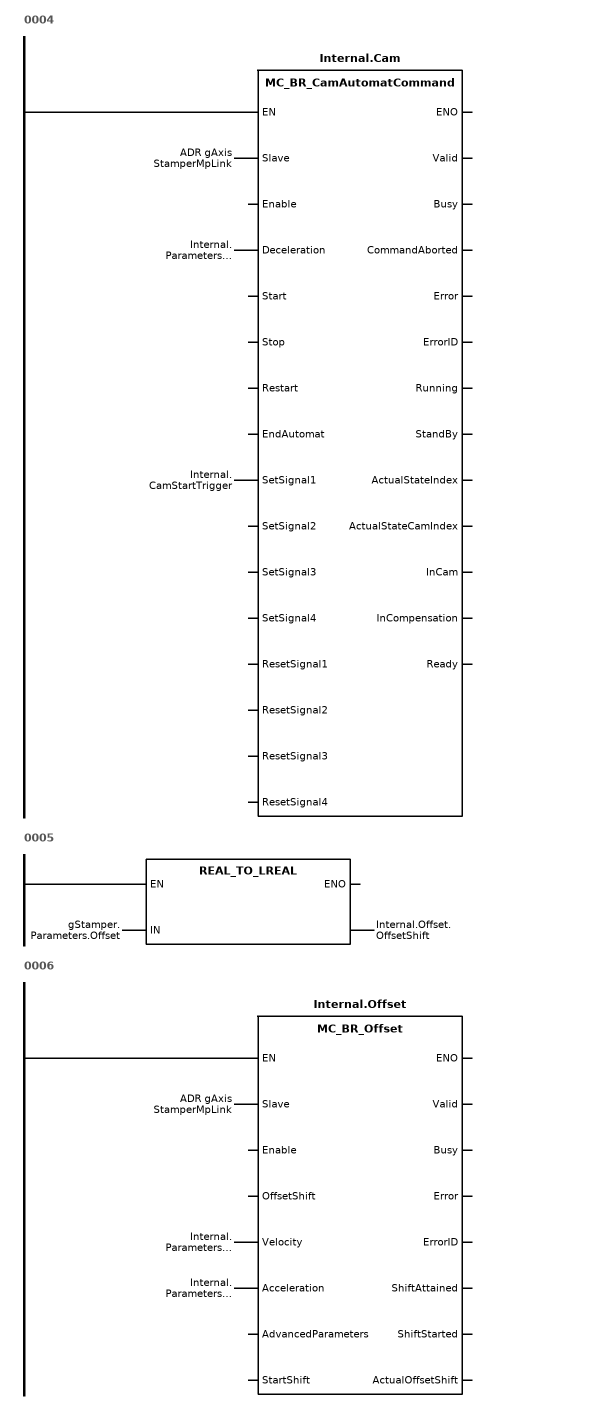
Ladder, written as Structured Text:
```iecst
ACTION MotionAction:
(* Network 1 *)
Internal.Parameters.Deceleration := gStamper.Parameters.Acceleration;

(* Network 2 *)
Internal.Parameters.Acceleration := gStamper.Parameters.Acceleration;

(* Network 3 *)
Internal.Axis(MpLink := ADR(gAxisStamperMpLink), Enable := gStamper.Commands.Enable, ErrorReset := gStamper.Commands.Reset, Parameters := ADR(Internal.Parameters));
gStamper.Interface.Outputs.SetPosition := Internal.Axis.Position;

(* Network 4 *)
Internal.Cam(Slave := ADR(gAxisStamperMpLink), Deceleration := Internal.Parameters.Deceleration, SetSignal1 := Internal.CamStartTrigger);

(* Network 5 *)
Internal.Offset.OffsetShift := REAL_TO_LREAL(gStamper.Parameters.Offset);

(* Network 6 *)
Internal.Offset(Slave := ADR(gAxisStamperMpLink), Velocity := Internal.Parameters.Velocity, Acceleration := Internal.Parameters.Acceleration);
END_ACTION
```

### MainMachineGlobalTypes.typ
```iecst
TYPE
	MainMachineType : 	STRUCT  (*MainMachine Main type*)
		Commands : MainMachineCommadsType;
		Feedbacks : MainMachineFeedbacksType;
		Parameters : MainMachineParametersType;
		Statistics : MainMachineStatisticsType;
	END_STRUCT;
	MainMachineCommadsType : 	STRUCT  (*MainMachine Commands type*)
		LinkMode : BOOL;
		Reset : BOOL;
		HeartBeat : BOOL;
		ClearStats : BOOL;
		Automatic : MainMachineAutomaticCommadsType;
		Manual : MainMachineManualCommadsType;
		OpcuaClientOk : BOOL;
	END_STRUCT;
	MainMachineFeedbacksType : 	STRUCT  (*MainMachine Feedbacks type*)
		WaitingStart : BOOL;
		Started : BOOL;
		Stopping : BOOL;
		Error : BOOL;
		HeartBeat : BOOL;
		AutomaticMode : BOOL;
		LinkOk : BOOL;
		ManualMode : BOOL;
		InitDone : BOOL;
		WaitModeSelection : BOOL;
		WaitingInit : BOOL;
		NewCapOnWork : BOOL;
		ClearStatsDone : BOOL;
		Initializing : BOOL;
		WaitingModulesReady : BOOL;
		PushingCap : BOOL;
		PickingCap : BOOL;
		DeliveringCap : BOOL;
		CapsOnConveyor : USINT;
		AskRemoveCaps : BOOL;
	END_STRUCT;
	MainMachineParametersType : 	STRUCT  (*MainMachine Parameters type*)
		StamperEnable : BOOL := TRUE;
	END_STRUCT;
	MainMachineStatisticsType : 	STRUCT
		CapsCounter : UDINT;
		CurrentCapWorkingTime : TIME;
		LastCapWorkingTime : TIME;
		AverageCapWorkingTime : TIME;
	END_STRUCT;
	MainMachineAutomaticCommadsType : 	STRUCT  (*MainMachine Commands type*)
		Enable : BOOL;
		Init : BOOL;
		Start : BOOL;
		CapsRemoved : BOOL;
	END_STRUCT;
	MainMachineManualCommadsType : 	STRUCT  (*MainMachine Commands type*)
		Enable : BOOL;
	END_STRUCT;
END_TYPE
```

### MainMachineGlobalVariables.var
```iecst
VAR
	gMainMachine : MainMachineType;
END_VAR
VAR CONSTANT
	STATS_HISTORY_MAX_INDEX : USINT := 9;
END_VAR
```

### Program Logical/Source/MainMachine/MainMachineProgram (IEC)

#### Main.st - Init, cyclic, exit code
```iecst
//******************************************************************************************************
// Program: 	MainMachineProgram
// Author: 		Andrea Pennisi
// Rev.: 		1.0.0
// Date:		5.12.2023
//
// Description:
// This module is the main machine. It manage the comunications between the modules and the working flow.
//******************************************************************************************************
PROGRAM _INIT

	EnableModules;

    MachineState.NextState := WAITING_MODE_SELECTION;

END_PROGRAM

PROGRAM _CYCLIC

	// Master communication management
	MasterCommunication;

	// Alarms
	SetAlarmsAction;

	// Check stop reaction
	IF MpAlarmXCheckReaction(gAlarmXCoreMpLink,'STOP') THEN
		MachineState.NextState := ERROR;
	END_IF

	// Machine state
	MachineStateManagementAction;
	CASE MachineState.ActualState OF

		WAITING_MODE_SELECTION:
			MachineState.TimeoutTimer.PT := T#0S; // Timeout disabled in this state
			IF MachineState.NewTriggerState THEN
				StopModules;
			END_IF

			IF gMainMachine.Commands.Automatic.Enable THEN
				MachineState.NextState := AUTO_WAITING_INIT;

			ELSIF gMainMachine.Commands.Manual.Enable THEN
				MachineState.NextState := MANUAL;
			END_IF

		MANUAL:
			MachineState.TimeoutTimer.PT := T#0S; // Timeout disabled in this state
			IF MachineState.NewTriggerState THEN
				ResetModulesManualCommands;
			END_IF

			gPusher.Commands.Manual.Enable := TRUE;
			gPicker.Commands.Manual.Enable := TRUE;
			gConveyor.Commands.Manual.Enable := TRUE;
			gStamper.Commands.Manual.Enable := TRUE;

			IF NOT gMainMachine.Commands.Manual.Enable THEN
				MachineState.NextState := WAITING_MODE_SELECTION;
			END_IF

		AUTO_WAITING_INIT:
			MachineState.TimeoutTimer.PT := T#0S; // Timeout disabled in this state
			IF MachineState.NewTriggerState THEN
				gMainMachine.Feedbacks.InitDone := FALSE;
			END_IF

			IF NOT gMainMachine.Commands.Automatic.Enable THEN
				MachineState.NextState := WAITING_MODE_SELECTION;

			ELSIF gMainMachine.Commands.Automatic.Init THEN
				MachineState.NextState := AUTO_INITIALIZING;

			END_IF

		AUTO_INITIALIZING:
			MachineState.TimeoutTimer.PT := T#30S; // Timeout disabled in this state
			IF MachineState.NewTriggerState THEN
				InitModules;
			END_IF

			IF gPusher.Feedbacks.InitDone
				AND gPicker.Feedbacks.InitDone
				AND gConveyor.Feedbacks.InitDone
				AND gStamper.Feedbacks.InitDone THEN

				gMainMachine.Feedbacks.InitDone := TRUE;
				MachineState.NextState := AUTO_WAITING_START;

			END_IF

		AUTO_WAITING_START:
			MachineState.TimeoutTimer.PT := T#0S; // Timeout disabled in this state
			IF MachineState.NewTriggerState THEN
				StopModules;
			END_IF

			IF NOT gMainMachine.Commands.Automatic.Enable THEN
				MachineState.NextState := WAITING_MODE_SELECTION;

			ELSIF gMainMachine.Commands.Automatic.Start THEN
				MachineState.NextState := AUTO_WAITING_MODULES_READY;

			ELSIF gMainMachine.Commands.Automatic.Init THEN
				gMainMachine.Feedbacks.InitDone := TRUE;

			END_IF

		AUTO_WAITING_MODULES_READY:
			MachineState.TimeoutTimer.PT := T#0S; // Timeout disabled in this state
			IF MachineState.NewTriggerState THEN
				StartModules;
				gMainMachine.Feedbacks.NewCapOnWork := FALSE;
			END_IF

			IF NOT gMainMachine.Commands.Automatic.Start THEN
				MachineState.NextState := WAITING_MODE_SELECTION;

			ELSIF gPusher.Feedbacks.WaitingTakeACapCommand
				AND gPicker.Feedbacks.WaitingPickCommand
				AND gConveyor.Feedbacks.WaitingCap
				AND (gStamper.Feedbacks.WaitingCap OR NOT gStamper.Commands.Automatic.Start) THEN

				MachineState.NextState := AUTO_PUSH_CAP;
			END_IF

		AUTO_PUSH_CAP:
			MachineState.TimeoutTimer.PT := T#0S; // Timeout disabled in this state
			IF MachineState.NewTriggerState THEN
				gMainMachine.Feedbacks.NewCapOnWork := TRUE;
				gPusher.Commands.Automatic.TakeACap := TRUE;
			END_IF

			IF NOT gPusher.Feedbacks.WaitingTakeACapCommand THEN
				gPusher.Commands.Automatic.TakeACap := FALSE;
			END_IF

			IF NOT gPusher.Commands.Automatic.TakeACap AND gPusher.Feedbacks.TakeACapDone THEN
				MachineState.NextState := AUTO_PICK_CAP;
			END_IF

		AUTO_PICK_CAP:
			MachineState.TimeoutTimer.PT := T#0S; // Timeout disabled in this state
			IF MachineState.NewTriggerState THEN
				gPicker.Commands.Automatic.PickACap := TRUE;
			END_IF

			IF NOT gPicker.Feedbacks.WaitingPickCommand THEN
				gPicker.Commands.Automatic.PickACap := FALSE;
			END_IF

			IF NOT gPicker.Commands.Automatic.PickACap AND gPicker.Feedbacks.PickACapDone THEN
				MachineState.NextState := AUTO_WAITING_CAP_DELIVERY;
			END_IF

		AUTO_WAITING_CAP_DELIVERY:
			MachineState.TimeoutTimer.PT := T#0S; // Timeout disabled in this state
			IF MachineState.NewTriggerState THEN
				gConveyor.Commands.Automatic.DeliverCap := TRUE;
				Internal.StamperOneTimeInterlock := FALSE;
			END_IF

			IF gConveyor.Feedbacks.CapsOnConveyor = 1 AND NOT Internal.StamperOneTimeInterlock THEN
				gStamper.Commands.Automatic.StampCap := TRUE;
				Internal.StamperOneTimeInterlock := TRUE;
			END_IF

			IF NOT gConveyor.Feedbacks.WaitingCap THEN
				gConveyor.Commands.Automatic.DeliverCap := FALSE;
			END_IF

			IF NOT gStamper.Feedbacks.WaitingCap THEN
				gStamper.Commands.Automatic.StampCap := FALSE;
			END_IF

			IF NOT gConveyor.Commands.Automatic.DeliverCap AND gConveyor.Feedbacks.DeliverCapDone THEN

				IF gStamper.Commands.Automatic.Start THEN

					IF NOT gStamper.Commands.Automatic.StampCap AND gStamper.Feedbacks.StampCapDone THEN
						MachineState.NextState := AUTO_WAITING_MODULES_READY;
					END_IF

				ELSE
					MachineState.NextState := AUTO_WAITING_MODULES_READY;
				END_IF

			END_IF

		ERROR:
			MachineState.TimeoutTimer.PT := T#0S; // Timeout disabled in this state
			IF MachineState.NewTriggerState THEN
				StopModules;
				ResetModulesManualCommands;
				gMainMachine.Commands.Reset := FALSE;
			END_IF

			IF EDGE(gMainMachine.Commands.Automatic.Init) THEN
				gMainMachine.Commands.Reset := gMainMachine.Commands.Automatic.Init; // User can reset alarms with init command
			END_IF

			gPusher.Commands.Reset := gMainMachine.Commands.Reset;
			gPicker.Commands.Reset := gMainMachine.Commands.Reset;
			gConveyor.Commands.Reset := gMainMachine.Commands.Reset;
			gStamper.Commands.Reset := gMainMachine.Commands.Reset;

			IF gMainMachine.Commands.Reset THEN
				gAlarms.MpAlarmXListUIConnect.AcknowledgeAll := TRUE;
			END_IF

			IF NOT MpAlarmXCheckReaction(gAlarmXCoreMpLink,'STOP') THEN

				gMainMachine.Commands.Reset := FALSE;
				MachineState.NextState := WAITING_MODE_SELECTION;
			END_IF

		ELSE
			MachineState.NextState := WAITING_MODE_SELECTION;

	END_CASE

	FeedbacksUpdateAction;

	StatisticsAction;

END_PROGRAM

PROGRAM _EXIT

END_PROGRAM
```

#### Types.typ - Local data types
```iecst
TYPE
	MachineStateType : 	STRUCT  (*Machine state main type*)
		OldState : MachineStateEnum; (*Actual state*)
		ActualState : MachineStateEnum; (*Actual state*)
		NextState : MachineStateEnum; (*Next state*)
		NewTriggerState : BOOL; (*Trigger state change*)
		TimeoutTimer : TON; (*State timeout*)
	END_STRUCT;
	MachineStateEnum :
		( (*Machine State enumeration*)
		WAITING_MODE_SELECTION,
		MANUAL,
		AUTO_WAITING_INIT,
		AUTO_INITIALIZING,
		AUTO_WAITING_START,
		AUTO_WAITING_MODULES_READY,
		AUTO_PUSH_CAP,
		AUTO_PICK_CAP,
		AUTO_WAITING_CAP_DELIVERY,
		ERROR (*ERROR state*)
		);
	InternalType : 	STRUCT
		HeartBeatTimer : TON := (PT:=T#250MS);
		CommunicationTimeoutTimer : TON := (PT:=T#3S);
		MasterCommunicationOk : BOOL;
		OnPhaseStopRequest : BOOL;
		Error : BOOL;
		StamperOneTimeInterlock : BOOL;
	END_STRUCT;
END_TYPE
```

#### Variables.var - Local variables
```iecst
VAR
	MachineState : MachineStateType;
	Internal : InternalType;
	CommunicationInitialized : BOOL;
	CapWorkStopwatch : TON := (PT:=T#24d);
	CapsWorkingTimeHistory : ARRAY[0..STATS_HISTORY_MAX_INDEX] OF TIME;
	TotHistoryWorkedTime : TIME;
	Index : USINT;
END_VAR
```

#### Actions.st
```iecst
ACTION FeedbacksUpdateAction:

	gMainMachine.Feedbacks.WaitingInit := MachineState.ActualState = AUTO_WAITING_INIT;

	gMainMachine.Feedbacks.Initializing := MachineState.ActualState = AUTO_INITIALIZING;

	gMainMachine.Feedbacks.WaitingStart := MachineState.ActualState = AUTO_WAITING_START;

	gMainMachine.Feedbacks.WaitingModulesReady := MachineState.ActualState = AUTO_WAITING_MODULES_READY;

	gMainMachine.Feedbacks.PushingCap := MachineState.ActualState = AUTO_PUSH_CAP;

	gMainMachine.Feedbacks.PickingCap := MachineState.ActualState = AUTO_PICK_CAP;

	gMainMachine.Feedbacks.DeliveringCap := MachineState.ActualState = AUTO_WAITING_CAP_DELIVERY;

	gMainMachine.Feedbacks.Error := MachineState.ActualState = ERROR;

	gMainMachine.Feedbacks.WaitModeSelection := MachineState.ActualState = WAITING_MODE_SELECTION;

	gMainMachine.Feedbacks.Stopping := gMainMachine.Feedbacks.Started AND Internal.OnPhaseStopRequest;

	gMainMachine.Feedbacks.ManualMode := (MachineState.ActualState = MANUAL);

	gMainMachine.Feedbacks.AutomaticMode := NOT gMainMachine.Feedbacks.ManualMode AND NOT gMainMachine.Feedbacks.WaitModeSelection AND NOT gMainMachine.Feedbacks.Error;

	gMainMachine.Feedbacks.CapsOnConveyor := gConveyor.Feedbacks.CapsOnConveyor;

	IF gMainMachine.Commands.Automatic.Init AND gMainMachine.Feedbacks.CapsOnConveyor > 0 THEN
		gMainMachine.Feedbacks.AskRemoveCaps := TRUE;
	ELSIF gMainMachine.Commands.Automatic.CapsRemoved THEN
		gMainMachine.Feedbacks.AskRemoveCaps := FALSE;
	END_IF

	// Started
	IF (MachineState.ActualState = AUTO_WAITING_MODULES_READY)
		OR (MachineState.ActualState = AUTO_PUSH_CAP)
		OR (MachineState.ActualState = AUTO_PICK_CAP)
		OR (MachineState.ActualState = AUTO_WAITING_CAP_DELIVERY) THEN

		gMainMachine.Feedbacks.Started := TRUE;
	ELSE
		gMainMachine.Feedbacks.Started := FALSE;
	END_IF

	IF NOT gMainMachine.Feedbacks.Started THEN
		gMainMachine.Feedbacks.NewCapOnWork := FALSE;
	END_IF

	IF NOT gMainMachine.Commands.Automatic.Init THEN
		gMainMachine.Feedbacks.InitDone := FALSE;
	END_IF
END_ACTION

ACTION MachineStateManagementAction:

    // Machine state timeout check
    MachineState.TimeoutTimer(IN := MachineState.TimeoutTimer.PT <> T#0S AND NOT MachineState.NewTriggerState);

	// Machine state change state logic
	MachineState.NewTriggerState := (MachineState.ActualState <> MachineState.NextState);
	IF MachineState.NewTriggerState THEN
		MachineState.OldState := MachineState.ActualState;
	END_IF
	MachineState.ActualState := MachineState.NextState;

END_ACTION

ACTION SetAlarmsAction:

	// Timeouts
	IF MachineState.TimeoutTimer.Q THEN

		// Throw here timeout alarms
		CASE MachineState.ActualState OF
		    AUTO_INITIALIZING: MpAlarmXSet(gAlarmXCoreMpLink,'MainMachineInitializationTimeout'); // Edge alarm!
		END_CASE

		MachineState.NextState := ERROR;
	END_IF

	// MainMachineEmergencyCircuitInterrupted
	IF FALSE THEN
		MpAlarmXSet(gAlarmXCoreMpLink,'MainMachineEmergencyCircuitInterrupted'); // Persistent alarm
	ELSE
		MpAlarmXReset(gAlarmXCoreMpLink,'MainMachineEmergencyCircuitInterrupted'); // Persistent alarm
	END_IF

	// MainMachineCommunicationLost
	IF NOT Internal.MasterCommunicationOk AND gMainMachine.Commands.LinkMode THEN
		MpAlarmXSet(gAlarmXCoreMpLink,'MainMachineCommunicationLost'); // Persistent alarm
	ELSE
		MpAlarmXReset(gAlarmXCoreMpLink,'MainMachineCommunicationLost'); // Persistent alarm
	END_IF

END_ACTION

ACTION MasterCommunication:

	// Send communication heart beat to the master
	Internal.HeartBeatTimer(IN:=NOT Internal.HeartBeatTimer.Q);
	IF Internal.HeartBeatTimer.Q THEN
		gMainMachine.Feedbacks.HeartBeat := NOT gMainMachine.Feedbacks.HeartBeat;
	END_IF

	// Check communication heart beat from the master
	IF EDGE(gMainMachine.Commands.HeartBeat) AND gMainMachine.Commands.OpcuaClientOk THEN
		Internal.CommunicationTimeoutTimer.IN := FALSE;
		CommunicationInitialized := TRUE;
	ELSE
		Internal.CommunicationTimeoutTimer.IN := TRUE;
		IF Internal.CommunicationTimeoutTimer.Q THEN
			CommunicationInitialized := TRUE;
		END_IF

	END_IF

	Internal.CommunicationTimeoutTimer();

	Internal.MasterCommunicationOk := NOT Internal.CommunicationTimeoutTimer.Q AND CommunicationInitialized;
	gMainMachine.Feedbacks.LinkOk := Internal.MasterCommunicationOk;

END_ACTION

ACTION EnableModules:

	gPusher.Commands.Enable := TRUE;

	gPicker.Commands.Enable := TRUE;

	gConveyor.Commands.Enable := TRUE;

	gStamper.Commands.Enable := TRUE;

END_ACTION

ACTION StopModules:

	gPusher.Commands.Manual.Enable := FALSE;
	gPusher.Commands.Automatic.Start := FALSE;
	gPusher.Commands.Automatic.Init := FALSE;
	gPusher.Commands.Reset := FALSE;
	gPusher.Commands.Automatic.TakeACap := FALSE;

	gPicker.Commands.Manual.Enable := FALSE;
	gPicker.Commands.Automatic.Start := FALSE;
	gPicker.Commands.Automatic.Init := FALSE;
	gPicker.Commands.Reset := FALSE;
	gPicker.Commands.Automatic.PickACap := FALSE;

	gConveyor.Commands.Manual.Enable := FALSE;
	gConveyor.Commands.Automatic.Start := FALSE;
	gConveyor.Commands.Automatic.Init := FALSE;
	gConveyor.Commands.Reset := FALSE;
	gConveyor.Commands.Automatic.DeliverCap := FALSE;

	gStamper.Commands.Manual.Enable := FALSE;
	gStamper.Commands.Automatic.Start := FALSE;
	gStamper.Commands.Automatic.Init := FALSE;
	gStamper.Commands.Reset := FALSE;
	gStamper.Commands.Automatic.StampCap := FALSE;

END_ACTION

ACTION ResetModulesManualCommands:

	memset(ADR(gPusher.Commands.Manual),0,SIZEOF(gPusher.Commands.Manual));
	memset(ADR(gPicker.Commands.Manual),0,SIZEOF(gPicker.Commands.Manual));
	memset(ADR(gConveyor.Commands.Manual),0,SIZEOF(gConveyor.Commands.Manual));
	memset(ADR(gStamper.Commands.Manual),0,SIZEOF(gStamper.Commands.Manual));

END_ACTION

ACTION InitModules:

	gPusher.Commands.Automatic.Init := TRUE;
	gPicker.Commands.Automatic.Init := TRUE;
	gConveyor.Commands.Automatic.Init := TRUE;
	gStamper.Commands.Automatic.Init := TRUE;

END_ACTION

ACTION StartModules:

	gPusher.Commands.Automatic.Start := TRUE;
	gPicker.Commands.Automatic.Start := TRUE;
	gConveyor.Commands.Automatic.Start := TRUE;
	gStamper.Commands.Automatic.Start := gMainMachine.Parameters.StamperEnable;

END_ACTION

ACTION StatisticsAction:

	// Stats clear
	IF gMainMachine.Commands.ClearStats THEN
		memset(ADR(CapsWorkingTimeHistory),0,SIZEOF(CapsWorkingTimeHistory));
		gMainMachine.Statistics.CapsCounter := 0;
		gMainMachine.Feedbacks.ClearStatsDone := TRUE;
		CapWorkStopwatch.IN := FALSE;
	ELSE
		gMainMachine.Feedbacks.ClearStatsDone := FALSE;
	END_IF

	// Manage the stopwatch to measure the current cap working time
	IF EDGE(gMainMachine.Feedbacks.NewCapOnWork) THEN
		IF gMainMachine.Feedbacks.NewCapOnWork THEN
			gMainMachine.Statistics.CapsCounter := gMainMachine.Statistics.CapsCounter + 1;
			CapWorkStopwatch.IN := TRUE;
		ELSE
			CapWorkStopwatch.IN := FALSE;
			memmove(ADR(CapsWorkingTimeHistory[1]),ADR(CapsWorkingTimeHistory[0]),SIZEOF(CapsWorkingTimeHistory)-SIZEOF(CapsWorkingTimeHistory[0]));
			CapsWorkingTimeHistory[0] := CapWorkStopwatch.ET;
		END_IF
	END_IF

	CapWorkStopwatch();

	// Calc the total amount of time stored in the history array
	TotHistoryWorkedTime := T#0S;
	FOR Index:=0 TO STATS_HISTORY_MAX_INDEX DO
		IF CapsWorkingTimeHistory[Index]>T#0s THEN
			TotHistoryWorkedTime := TotHistoryWorkedTime + CapsWorkingTimeHistory[Index];
		ELSE
			EXIT;
		END_IF
	END_FOR

	gMainMachine.Statistics.CurrentCapWorkingTime := CapWorkStopwatch.ET;
	gMainMachine.Statistics.LastCapWorkingTime := CapsWorkingTimeHistory[0];
	gMainMachine.Statistics.AverageCapWorkingTime := UDINT_TO_TIME(TIME_TO_UDINT(TotHistoryWorkedTime)/MAX(1,Index));
END_ACTION
```

### HMIGlobalTypes.typ
```iecst
TYPE
	HMIType : 	STRUCT  (*HMI Main type*)
		AutomaticPage : HMIAutomaticPageType;
		ManualPage : HMIManualPageType;
		HeaderContent : HMIHeaderContentType;
	END_STRUCT;
	HMIAutomaticPageType : 	STRUCT  (*HMI Interface Output type*)
		StartButtonEnable : BOOL;
		StartButton : BOOL;
		StopButtonVisibility : BOOL;
		InitButtonEnable : BOOL;
		InitButton : BOOL;
		ConveyorSpeed : REAL;
		ConveyorSpeedEnable : BOOL;
		AutoButtonEnable : BOOL;
		AutoButton : BOOL;
		LinkButtonEnable : BOOL;
		LinkButton : BOOL;
		ReadyToStartVisibility : BOOL;
		CurrentCapWorkingTime : UDINT;
		LastCapWorkedTime : UDINT;
		AvgCapWorkTime : UDINT;
		ClearStats : BOOL;
		StamperIncludedCheckbox : BOOL;
		StamperIncludedCheckboxEnable : BOOL;
		StamperOffset : REAL;
		StamperOffsetEnable : BOOL;
		CapsCounter : UDINT;
		AskRemoveCaps : BOOL;
		CapsRemoved : BOOL;
	END_STRUCT;
	HMIManualPageType : 	STRUCT  (*HMI Interface Output type*)
		ManualButtonEnable : BOOL;
		ManualButton : BOOL;
		PushCapButtonEnable : BOOL;
		PushCapButton : BOOL;
		ArmForwardButtonEnable : BOOL;
		ArmForwardButton : BOOL;
		ArmBackwardButtonEnable : BOOL;
		ArmBackwardButton : BOOL;
		ArmVaacumButtonEnable : BOOL;
		ArmVaacumButton : BOOL;
		ConveyorHomeButtonEnable : BOOL;
		ConveyorHomeButton : BOOL;
		ConveyorPowerButtonEnable : BOOL;
		ConveyorPowerButton : BOOL;
		ConveyorMoveButtonEnable : BOOL;
		ConveyorMoveButton : BOOL;
		ConveyorSpeed : REAL;
		ConveyorSpeedEnable : BOOL;
		ConveyorAxisHomed : BOOL;
		ConveyorAxisPowered : BOOL;
		StamperHomeButtonEnable : BOOL;
		StamperHomeButton : BOOL;
		StamperPowerButtonEnable : BOOL;
		StamperPowerButton : BOOL;
		StamperMoveButtonEnable : BOOL;
		StamperMoveButton : BOOL;
		StamperSpeed : REAL;
		StamperSpeedEnable : BOOL;
		StamperAxisHomed : BOOL;
		StamperAxisPowered : BOOL;
		StamperForwardButtonEnable : BOOL;
		StamperForwardButton : BOOL;
		StamperPosition : LREAL;
		StamperPositionEnable : BOOL;
		PusherInterface : PusherInterfaceType;
		PickerInterface : PickerInterfaceType;
		ConveyorInterface : ConveyorInterfaceType;
		StamperInterface : StamperInterfaceType;
		ConveyorActSpeed : REAL;
		ConveyorActPosition : LREAL;
		StamperActSpeed : REAL;
		StamperActPosition : LREAL;
		ConveyorAcceleration : REAL;
		ConveyorAccelerationEnable : BOOL;
		StamperAcceleration : REAL;
		StamperAccelerationEnable : BOOL;
	END_STRUCT;
	HMIHeaderContentType : 	STRUCT  (*HMI Interface Output type*)
		MasterConnectionOk : BOOL;
		PendingAlarms : STRING[3];
		StateManual : BOOL;
		StateWaitingInit : BOOL;
		StateInitializing : BOOL;
		StateWaitingStart : BOOL;
		StateWaitingModulesReady : BOOL;
		StatePushingCap : BOOL;
		StatePickingCap : BOOL;
		StateDeliveringCap : BOOL;
		StateError : BOOL;
		StateWaitModeSelection : BOOL;
		ResetAlarms : BOOL;
		AlarmBlink : BOOL;
	END_STRUCT;
END_TYPE
```

### HMIGlobalVariables.var
```iecst
VAR
    gHMI : HMIType;
END_VAR
```

### Program Logical/Source/HMI/HMIProgram (IEC)

#### Main.st - Init, cyclic, exit code
```iecst
//******************************************************************************************************
// Program: 	HMIProgram
// Author: 		Andrea Pennisi
// Rev.: 		1.0.0
// Date:		5.12.2023
//
// Description:
// This module is used to manage the enables/visibility and value of the variable in the HMI
//******************************************************************************************************
PROGRAM _INIT
	SetInitialValuesAction;
END_PROGRAM

PROGRAM _CYCLIC

	HeaderContentAction;

	AutomaticPageAction;

	ManualPageAction;

END_PROGRAM

PROGRAM _EXIT

END_PROGRAM
```

#### Variables.var - Local variables
```iecst
VAR
	AlarmBlinkTimer : TON;
END_VAR
```
